FUNCTION_BLOCK "CompValEqOr"   // FB55, LAD
TITLE = COMP_VAL_==_OR_FB / COMP_VAL_==_OR
AUTHOR : SICAR
FAMILY : Miscellaneous
VERSION : 1.0
// Der Baustein vergleicht die Werte der Eingänge in1...in8 mit dem Wert des Eingangs „compareValue“ und verodert diese Vergleiche. Ist mindestens einer der Werte von in1...in8 gleich mit „compareValue“, so wird der Wert von „compareValue“ in den Output „value“ geschrieben. Andernfalls wird er mit dem Wert 0 beschrieben.  
// Anwendungsfall Beispiel: Damit kann ein "Summensignal" gebildet werden, z.B. für Produktionsdaten "Grenzwerte", womit ein Button animiert werden kann (Button "ProdData", "Grenzwerte").  
// 
// **Beispielaufruf**  
// Abbildung in Kontaktplan (KOP), ohne Parameterbeschaltung.  
// 
// **Aufrufschnittstelle**  
// Der Baustein wird im zyklischen Programm aufgerufen. In den Startup-Projekten ist der Baustein aufgerufen, für die Bildung eines Sammelsignals für die Grenzwerte der Produktionsdaten. Damit werden die Buttons  [ProdData]
// Compare the values of the inputs with the value of th input _compareValue_ generating a collective OR signal from these comparisons.
// stored: IsIECCheckEnabled true, MemoryReserve 100, SetENOAutomatically true
   VAR_INPUT
      compareValue { ExternalAccessible := 'False'; ExternalVisible := 'False'; ExternalWritable := 'False'} : UInt;   // Vergleichs Wert / Compare value
      val1 { ExternalAccessible := 'False'; ExternalVisible := 'False'; ExternalWritable := 'False'} : UInt;   // Wert 1 / value 1
      val2 { ExternalAccessible := 'False'; ExternalVisible := 'False'; ExternalWritable := 'False'} : UInt;   // Wert 2 / value 2
      val3 { ExternalAccessible := 'False'; ExternalVisible := 'False'; ExternalWritable := 'False'} : UInt;   // Wert 3 / value 3
      val4 { ExternalAccessible := 'False'; ExternalVisible := 'False'; ExternalWritable := 'False'} : UInt;   // Wert 4 / value 4
      val5 { ExternalAccessible := 'False'; ExternalVisible := 'False'; ExternalWritable := 'False'} : UInt;   // Wert 5 / value 5
      val6 { ExternalAccessible := 'False'; ExternalVisible := 'False'; ExternalWritable := 'False'} : UInt;   // Wert 6 / value 6
      val7 { ExternalAccessible := 'False'; ExternalVisible := 'False'; ExternalWritable := 'False'} : UInt;   // Wert 7 / value 7
      val8 { ExternalAccessible := 'False'; ExternalVisible := 'False'; ExternalWritable := 'False'} : UInt;   // Wert 8 / value 8
   END_VAR
   VAR_OUTPUT
      value { ExternalAccessible := 'False'; ExternalVisible := 'False'; ExternalWritable := 'False'} : UInt;   // Ergebnis Wert / Result value
   END_VAR
   VAR_TEMP
      tempDummy : Bool;   // Dummy
   END_VAR
BEGIN

REGION Network 1: Aufruf: Initialisierung SPS / ChangeLog
   // SIEMENS AG / (c)Copyright 2023
   // ------------------------------------------------------------------------------
   // Title:            CompValEqOr (FB55)
   // Comment/Function: Compare the values of the inputs with the value of th input compareValue generating a collective OR signal from these comparisons.
   // Library/Family:   Automation Framework
   // Author:           Siemens Digital Industry
   // Tested with:      ---
   // Engineering:      TIA Portal V19
   // Restrictions:     -
   // Requirements:     ---
   // ------------------------------------------------------------------------------
   // Change log table:
   // Version  | Date       | Expert in charge       | Changes applied
   // ---------|------------|------------------------|------------------------------
   // 01.00.00 | 11.12.2023 | Siemens Industry Online Support
   //                         First released version
END_REGION

REGION Network 2: Beschreibung / Description
   // The block compares the values of the inputs _in1 ... in8_ with the value of the input _compareValue_ and generates a collective OR signal from these comparisons. If at least one of the values of in1 ... in8 is equal with _compareValue_, the value of _compareValue_ is written to output “value”.  
   // Otherwise, “value” is written with the value 0.  
   // Use Case example: With this, a "summary signal" can be formed, e.g. for production data "Limit Values", with which a button can be animated (Button "ProdData", "LimitValues"). 
   // 
   // **Block call example**  
   // 
   // The call is shown as “Ladder Diagram” (LAD), without parameters.  
   // 
   // **Calling interface**  
   // 
   // The block is called in the cyclic program. In the startup projects, the block is called to generate a collective signal for the limit values of the production data. The buttons [ProdData] and [LimitValues] are animated in color, depending on the value range of the limit values.
   // 
   // **Operation mode Automatic / Manual**  
   // 
   // The block is independent of operation modes. Therefor it is not assigned to any operation mode area.
END_REGION

REGION Network 3: VALUE = 0 schreiben / set VALUE = 0
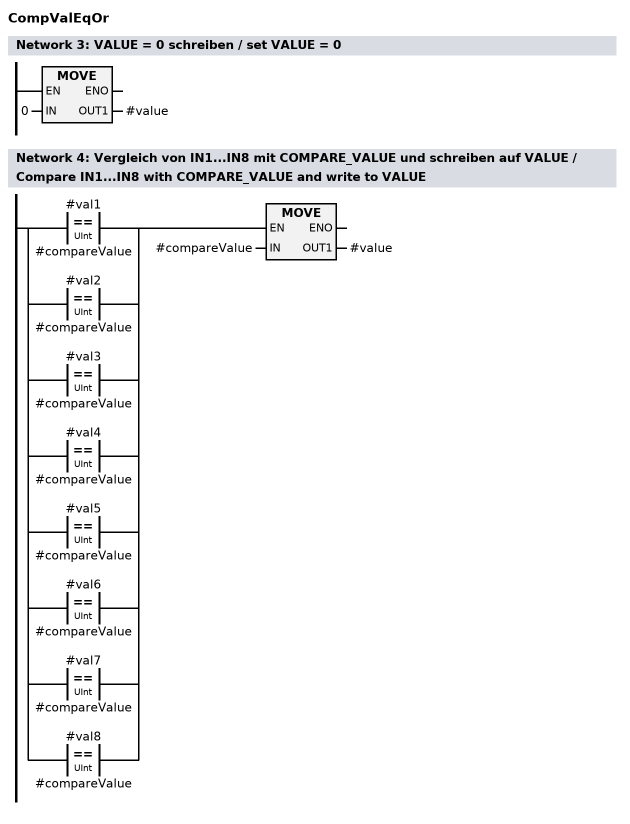
   RUNG wire#powerrail
      Move(in := 0, out1 => #value)
   END_RUNG
   // the same network as SCL:
   #value := 0;
END_REGION

REGION Network 4: Vergleich von IN1...IN8 mit COMPARE_VALUE und schreiben auf VALUE / Compare IN1...IN8 with COMPARE_VALUE and write to VALUE
   RUNG wire#powerrail
      { S7_Templates := "SrcType := UInt" } EQ_Contact(in1 := #val1, in2 := #compareValue)
      wire#w1
      Move(in := #compareValue, out1 => #value)
   END_RUNG
   RUNG wire#powerrail
      { S7_Templates := "SrcType := UInt" } EQ_Contact(in1 := #val2, in2 := #compareValue)
   END_RUNG wire#w1
   RUNG wire#powerrail
      { S7_Templates := "SrcType := UInt" } EQ_Contact(in1 := #val3, in2 := #compareValue)
   END_RUNG wire#w1
   RUNG wire#powerrail
      { S7_Templates := "SrcType := UInt" } EQ_Contact(in1 := #val4, in2 := #compareValue)
   END_RUNG wire#w1
   RUNG wire#powerrail
      { S7_Templates := "SrcType := UInt" } EQ_Contact(in1 := #val5, in2 := #compareValue)
   END_RUNG wire#w1
   RUNG wire#powerrail
      { S7_Templates := "SrcType := UInt" } EQ_Contact(in1 := #val6, in2 := #compareValue)
   END_RUNG wire#w1
   RUNG wire#powerrail
      { S7_Templates := "SrcType := UInt" } EQ_Contact(in1 := #val7, in2 := #compareValue)
   END_RUNG wire#w1
   RUNG wire#powerrail
      { S7_Templates := "SrcType := UInt" } EQ_Contact(in1 := #val8, in2 := #compareValue)
   END_RUNG wire#w1
   // the same network as SCL:
   IF (#val1 = #compareValue) OR (#val2 = #compareValue) OR (#val3 = #compareValue) OR (#val4 = #compareValue) OR (#val5 = #compareValue) OR (#val6 = #compareValue) OR (#val7 = #compareValue) OR (#val8 = #compareValue) THEN
       #value := #compareValue;
   END_IF;
END_REGION
END_FUNCTION_BLOCK

FUNCTION_BLOCK "CallAlarmCounter"   // FB5, LAD
// stored: MemoryReserve 100, SetENOAutomatically false
   VAR
      statPulse { ExternalAccessible := 'False'; ExternalVisible := 'False'; ExternalWritable := 'False'} : Array[0..99] of Bool;
   END_VAR
   VAR_TEMP
      tempEnter : Bool;   // Enter the conditions for the count to increase.
   END_VAR
   VAR_TEMP   // added for the SCL form of the ladder/FBD networks
      _w1 : Bool;
   END_VAR
BEGIN

REGION Network 1: Counter Setting Save
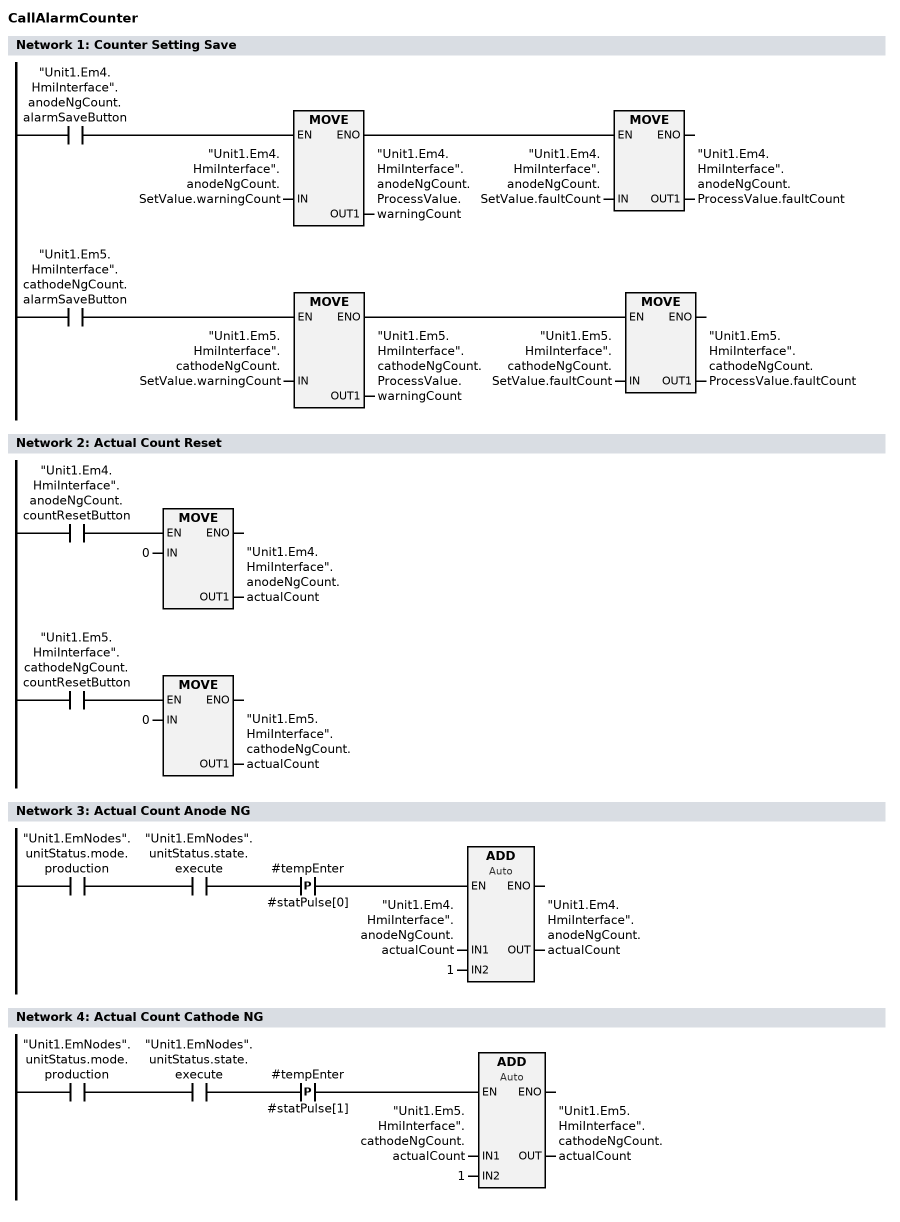
   RUNG wire#powerrail
      Contact( "Unit1.Em4.HmiInterface".anodeNgCount.alarmSaveButton )
      Move(in := "Unit1.Em4.HmiInterface".anodeNgCount.SetValue.warningCount, out1 => "Unit1.Em4.HmiInterface".anodeNgCount.ProcessValue.warningCount)
      Move(in := "Unit1.Em4.HmiInterface".anodeNgCount.SetValue.faultCount, out1 => "Unit1.Em4.HmiInterface".anodeNgCount.ProcessValue.faultCount)
   END_RUNG
   RUNG wire#powerrail
      Contact( "Unit1.Em5.HmiInterface".cathodeNgCount.alarmSaveButton )
      Move(in := "Unit1.Em5.HmiInterface".cathodeNgCount.SetValue.warningCount, out1 => "Unit1.Em5.HmiInterface".cathodeNgCount.ProcessValue.warningCount)
      Move(in := "Unit1.Em5.HmiInterface".cathodeNgCount.SetValue.faultCount, out1 => "Unit1.Em5.HmiInterface".cathodeNgCount.ProcessValue.faultCount)
   END_RUNG
   // the same network as SCL:
   IF "Unit1.Em4.HmiInterface".anodeNgCount.alarmSaveButton THEN
       "Unit1.Em4.HmiInterface".anodeNgCount.ProcessValue.warningCount := "Unit1.Em4.HmiInterface".anodeNgCount.SetValue.warningCount;
       "Unit1.Em4.HmiInterface".anodeNgCount.ProcessValue.faultCount := "Unit1.Em4.HmiInterface".anodeNgCount.SetValue.faultCount;
   END_IF;
   IF "Unit1.Em5.HmiInterface".cathodeNgCount.alarmSaveButton THEN
       "Unit1.Em5.HmiInterface".cathodeNgCount.ProcessValue.warningCount := "Unit1.Em5.HmiInterface".cathodeNgCount.SetValue.warningCount;
       "Unit1.Em5.HmiInterface".cathodeNgCount.ProcessValue.faultCount := "Unit1.Em5.HmiInterface".cathodeNgCount.SetValue.faultCount;
   END_IF;
END_REGION

REGION Network 2: Actual Count Reset
   RUNG wire#powerrail
      Contact( "Unit1.Em4.HmiInterface".anodeNgCount.countResetButton )
      Move(in := 0, out1 => "Unit1.Em4.HmiInterface".anodeNgCount.actualCount)
   END_RUNG
   RUNG wire#powerrail
      Contact( "Unit1.Em5.HmiInterface".cathodeNgCount.countResetButton )
      Move(in := 0, out1 => "Unit1.Em5.HmiInterface".cathodeNgCount.actualCount)
   END_RUNG
   // the same network as SCL:
   IF "Unit1.Em4.HmiInterface".anodeNgCount.countResetButton THEN
       "Unit1.Em4.HmiInterface".anodeNgCount.actualCount := 0;
   END_IF;
   IF "Unit1.Em5.HmiInterface".cathodeNgCount.countResetButton THEN
       "Unit1.Em5.HmiInterface".cathodeNgCount.actualCount := 0;
   END_IF;
END_REGION

REGION Network 3: Actual Count Anode NG
   RUNG wire#powerrail
      Contact( "Unit1.EmNodes".unitStatus.mode.production )
      Contact( "Unit1.EmNodes".unitStatus.state.execute )
      P_Contact(operand := #tempEnter, bit := #statPulse[0])
      Add(in1 := "Unit1.Em4.HmiInterface".anodeNgCount.actualCount, in2 := 1, out => "Unit1.Em4.HmiInterface".anodeNgCount.actualCount)
   END_RUNG
   // the same network as SCL:
   #_w1 := "Unit1.EmNodes".unitStatus.mode.production AND "Unit1.EmNodes".unitStatus.state.execute AND #tempEnter AND NOT #statPulse[0];   // rising edge of #tempEnter
   #statPulse[0] := #tempEnter;
   IF #_w1 THEN
       "Unit1.Em4.HmiInterface".anodeNgCount.actualCount := "Unit1.Em4.HmiInterface".anodeNgCount.actualCount + 1;
   END_IF;
END_REGION

REGION Network 4: Actual Count Cathode NG
   RUNG wire#powerrail
      Contact( "Unit1.EmNodes".unitStatus.mode.production )
      Contact( "Unit1.EmNodes".unitStatus.state.execute )
      P_Contact(operand := #tempEnter, bit := #statPulse[1])
      Add(in1 := "Unit1.Em5.HmiInterface".cathodeNgCount.actualCount, in2 := 1, out => "Unit1.Em5.HmiInterface".cathodeNgCount.actualCount)
   END_RUNG
   // the same network as SCL:
   #_w1 := "Unit1.EmNodes".unitStatus.mode.production AND "Unit1.EmNodes".unitStatus.state.execute AND #tempEnter AND NOT #statPulse[1];   // rising edge of #tempEnter
   #statPulse[1] := #tempEnter;
   IF #_w1 THEN
       "Unit1.Em5.HmiInterface".cathodeNgCount.actualCount := "Unit1.Em5.HmiInterface".cathodeNgCount.actualCount + 1;
   END_IF;
END_REGION
END_FUNCTION_BLOCK

FUNCTION "CallSettings" : Void   // FC8, LAD
// Call of settings blocks
// stored: IsIECCheckEnabled true, SetENOAutomatically false
BEGIN

REGION Network 1: Beschreibung / BLOCK INFO HEADER
   // **Betriebsart Automatik / Hand**  
   // Der Baustein ist keiner Betriebsart / Betriebsartenbereich zugeordnet.  
   // 
   // **Alarme**  
   // Der Baustein generiert keine Alarme.  
   // 
   // #### PLC-Datentypen  
   // Verwendete PLC-Datentypen für den SPS-Programmbaustein und das zugehörige WinCC-Bild.  
   // 
   // {.pageWidth}
   // ![Image](CallInterfaceSignals/de/image1.PNG)
   //  
   //  
   // #### Bausteinaufrufe 
   // Der Baustein “LSicar_InterfaceSignalsBool“ wird in diesem FB als Multi-Instanz aufgerufen, entspr. nebenstehender beispielhafter Darstellung.  
   // 
   // {.pageWidth}
   // ![Image](CallInterfaceSignals/de/image2.PNG)
   //  
   // Um einen neuen FB aufzurufen, ziehen Sie den FB in ein neues Netzwerk, wählen Sie „Multiinstanz“ aus, vergeben Sie einen Namen und parametrieren Sie den FB-Aufruf.  
   // 
   // {.pageWidth}
   // ![Image](CallInterfaceSignals/de/image3.PNG)
   //  
   //  
   // #### Weitere Hinweise 
   // 
   // #### Updateinfo 
   // 
   // #### Weitere Dokumente 
   // 
   // ![Icon](_Icon/reference.PNG)
   // 
   // ..\Library Types\LSicar_InterfaceSignalsBool.pdf
   // SIEMENS AG / (c)Copyright 2023
   // ------------------------------------------------------------------------------
   // Title:            CallSettings
   // Comment/Function: Call of SICAR Settings blocks
   // Library/Family:   -
   // Author:           -
   // Tested with:      ---
   // Engineering:      TIA Portal V19
   // Restrictions:     -
   // Requirements:     ---
   // ------------------------------------------------------------------------------
   // Change log table:
   // Version | Date | Expert in charge | Changes applied
   // -------|---------|-------------|--------------------------------------------
   // 01.00.00 | 01.01.1999 | Person x | First released version
   // 01.00.01 | 02.01.1999 | Person y | Block was Updated
END_REGION

REGION Network 2: Set set PLC date and time
   // Change local date and time of the PLC
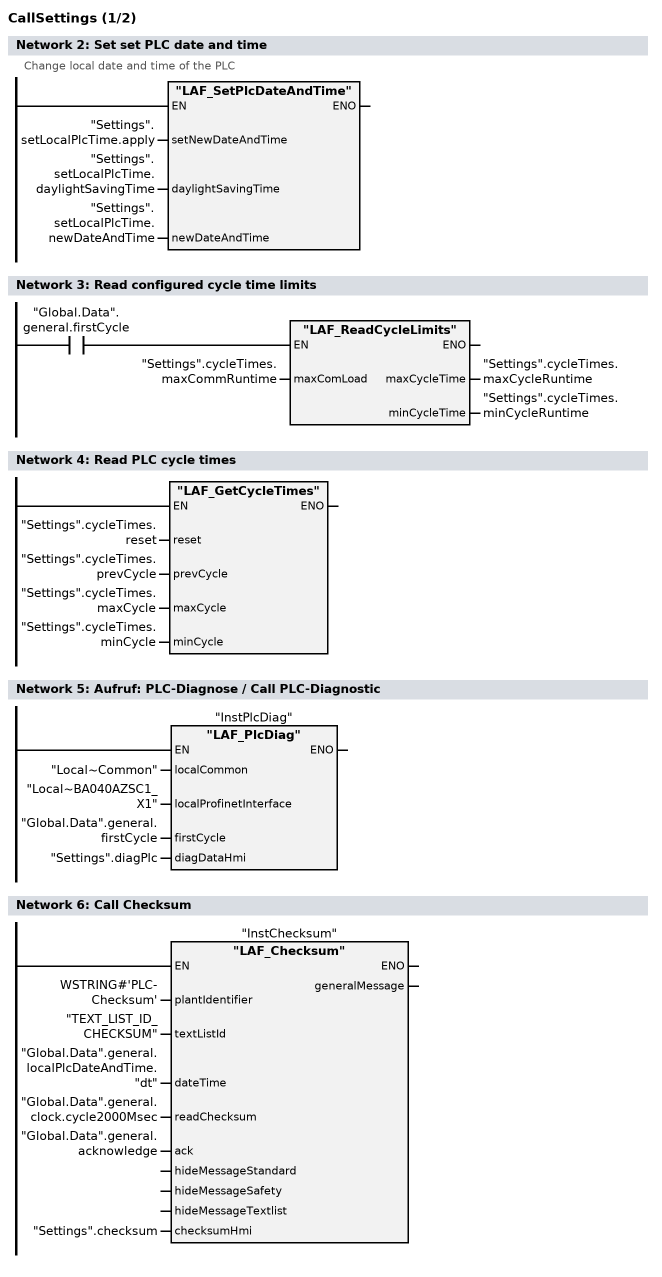
   RUNG wire#powerrail
      "LAF_SetPlcDateAndTime"(setNewDateAndTime := "Settings".setLocalPlcTime.apply, daylightSavingTime := "Settings".setLocalPlcTime.daylightSavingTime, newDateAndTime := "Settings".setLocalPlcTime.newDateAndTime)
   END_RUNG
   // the same network as SCL:
   "LAF_SetPlcDateAndTime"(setNewDateAndTime := "Settings".setLocalPlcTime.apply,
                           daylightSavingTime := "Settings".setLocalPlcTime.daylightSavingTime,
                           newDateAndTime := "Settings".setLocalPlcTime.newDateAndTime);
END_REGION

REGION Network 3: Read configured cycle time limits
   RUNG wire#powerrail
      Contact( "Global.Data".general.firstCycle )
      "LAF_ReadCycleLimits"(maxComLoad := "Settings".cycleTimes.maxCommRuntime, maxCycleTime => "Settings".cycleTimes.maxCycleRuntime, minCycleTime => "Settings".cycleTimes.minCycleRuntime)
   END_RUNG
   // the same network as SCL:
   IF "Global.Data".general.firstCycle THEN
       "LAF_ReadCycleLimits"(maxComLoad := "Settings".cycleTimes.maxCommRuntime,
                             maxCycleTime => "Settings".cycleTimes.maxCycleRuntime,
                             minCycleTime => "Settings".cycleTimes.minCycleRuntime);
   END_IF;
END_REGION

REGION Network 4: Read PLC cycle times
   RUNG wire#powerrail
      "LAF_GetCycleTimes"(reset := "Settings".cycleTimes.reset, prevCycle := "Settings".cycleTimes.prevCycle, maxCycle := "Settings".cycleTimes.maxCycle, minCycle := "Settings".cycleTimes.minCycle)
   END_RUNG
   // the same network as SCL:
   "LAF_GetCycleTimes"(reset := "Settings".cycleTimes.reset,
                       prevCycle := "Settings".cycleTimes.prevCycle,
                       maxCycle := "Settings".cycleTimes.maxCycle,
                       minCycle := "Settings".cycleTimes.minCycle);
END_REGION

REGION Network 5: Aufruf: PLC-Diagnose / Call PLC-Diagnostic
   RUNG wire#powerrail
      "InstPlcDiag"(localCommon := "Local~Common", localProfinetInterface := "Local~BA040AZSC1_X1", firstCycle := "Global.Data".general.firstCycle, diagDataHmi := "Settings".diagPlc)
   END_RUNG
   // the same network as SCL:
   "InstPlcDiag"(localCommon := "Local~Common",   // "LAF_PlcDiag"
                 localProfinetInterface := "Local~BA040AZSC1_X1",
                 firstCycle := "Global.Data".general.firstCycle,
                 diagDataHmi := "Settings".diagPlc);
END_REGION

REGION Network 6: Call Checksum
   RUNG wire#powerrail
      "InstChecksum"(plantIdentifier := WSTRING#'PLC-Checksum', textListId := "TEXT_LIST_ID_CHECKSUM", dateTime := "Global.Data".general.localPlcDateAndTime."dt", readChecksum := "Global.Data".general.clock.cycle2000Msec, ack := "Global.Data".general.acknowledge, hideMessageStandard :=, hideMessageSafety :=, hideMessageTextlist :=, checksumHmi := "Settings".checksum, generalMessage =>)
   END_RUNG
   // the same network as SCL:
   "InstChecksum"(plantIdentifier := WSTRING#'PLC-Checksum',   // "LAF_Checksum"
                  textListId := "TEXT_LIST_ID_CHECKSUM",
                  dateTime := "Global.Data".general.localPlcDateAndTime."dt",
                  readChecksum := "Global.Data".general.clock.cycle2000Msec,
                  ack := "Global.Data".general.acknowledge,
                  checksumHmi := "Settings".checksum);
END_REGION

REGION Network 7: Aufruf: SMC-Diagnose (SIMATIC Memory Card - Diagnose) / Call SMC-Diagnostic (SIMATIC Memory Card - Diagnostic)
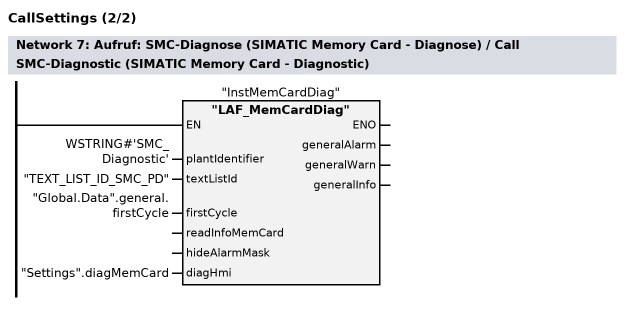
   RUNG wire#powerrail
      "InstMemCardDiag"(plantIdentifier := WSTRING#'SMC_Diagnostic', textListId := "TEXT_LIST_ID_SMC_PD", firstCycle := "Global.Data".general.firstCycle, readInfoMemCard :=, hideAlarmMask :=, diagHmi := "Settings".diagMemCard, generalAlarm =>, generalWarn =>, generalInfo =>)
   END_RUNG
   // the same network as SCL:
   "InstMemCardDiag"(plantIdentifier := WSTRING#'SMC_Diagnostic',   // "LAF_MemCardDiag"
                     textListId := "TEXT_LIST_ID_SMC_PD",
                     firstCycle := "Global.Data".general.firstCycle,
                     diagHmi := "Settings".diagMemCard);
END_REGION
END_FUNCTION

FUNCTION "CallEnergy" : Void   // FC5, LAD
TITLE = CallEnergy
// Call of Demo EnergyMeter and Energy Efficient M for EEMM demonstration
// stored: IsIECCheckEnabled true, SetENOAutomatically true
BEGIN

REGION Network 1: BLOCK INFO HEADER
   // SIEMENS AG / (c)Copyright 2023
   // ------------------------------------------------------------------------------
   // Title:            CallEnergy (FC5)
   // Comment/Function: Call of Demo EnergyMeter and Energy Efficient M for EEMM demonstration
   // Library/Family:   Energy
   // Author:           SICAR
   // Tested with:      ---
   // Engineering:      TIA Portal V19
   // Restrictions:     -
   // Requirements:     ---
   // ------------------------------------------------------------------------------
   // Change log table:
   // Version  | Date       | Expert in charge       | Changes applied
   // ---------|------------|------------------------|------------------------------
   // 01.00.00 | 11.12.2023 | SICAR
   //                         First released version
END_REGION

REGION Network 2: Call: Demo EnergyMeter, Energy Efficient M
   // Call for EEM demonstration
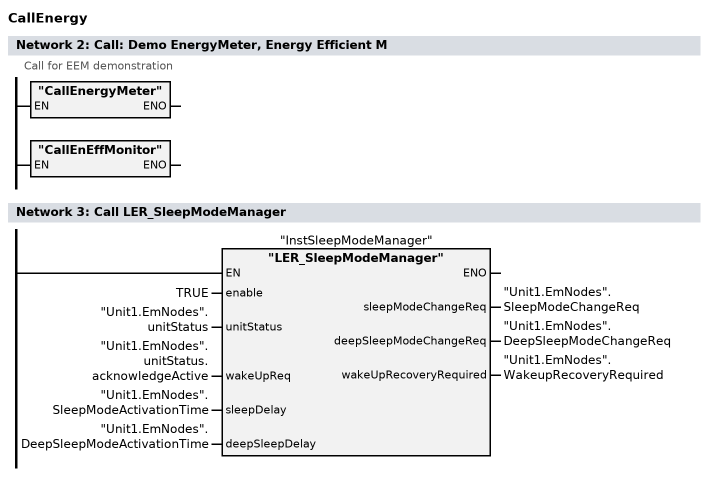
   RUNG wire#powerrail
      "CallEnergyMeter"()
   END_RUNG
   RUNG wire#powerrail
      "CallEnEffMonitor"()
   END_RUNG
   // the same network as SCL:
   "CallEnergyMeter"();
   "CallEnEffMonitor"();
END_REGION

REGION Network 3: Call LER_SleepModeManager
   RUNG wire#powerrail
      "InstSleepModeManager"(enable := TRUE, unitStatus := "Unit1.EmNodes".unitStatus, wakeUpReq := "Unit1.EmNodes".unitStatus.acknowledgeActive, sleepDelay := "Unit1.EmNodes".SleepModeActivationTime, deepSleepDelay := "Unit1.EmNodes".DeepSleepModeActivationTime, sleepModeChangeReq => "Unit1.EmNodes".SleepModeChangeReq, deepSleepModeChangeReq => "Unit1.EmNodes".DeepSleepModeChangeReq, wakeUpRecoveryRequired => "Unit1.EmNodes".WakeupRecoveryRequired)
   END_RUNG
   // the same network as SCL:
   "InstSleepModeManager"(enable := TRUE,   // "LER_SleepModeManager"
                          unitStatus := "Unit1.EmNodes".unitStatus,
                          wakeUpReq := "Unit1.EmNodes".unitStatus.acknowledgeActive,
                          sleepDelay := "Unit1.EmNodes".SleepModeActivationTime,
                          deepSleepDelay := "Unit1.EmNodes".DeepSleepModeActivationTime,
                          sleepModeChangeReq => "Unit1.EmNodes".SleepModeChangeReq,
                          deepSleepModeChangeReq => "Unit1.EmNodes".DeepSleepModeChangeReq,
                          wakeUpRecoveryRequired => "Unit1.EmNodes".WakeupRecoveryRequired);
END_REGION
END_FUNCTION

FUNCTION "CallEnergyMeter" : Void   // FC9, LAD
TITLE = CALL_AIEnergyMeter_FC
AUTHOR : SICAR
FAMILY : Energy
VERSION : 1.0
// FUNKTIONSBESCHREIBUNG: 
// Der Baustein dient als Aufrufschnittstelle für die bausteine des AI-Energy-Managements.
// Weitere Hinweise: siehe SICAR anwenderdefinierte Dokumentation / SICAR Online-Hilfe.
// This block calls the blocks for the AI-Energy-management.
// For more informations see SICAR userdefined documentation / SICAR online-help.
// stored: IsIECCheckEnabled true, SetENOAutomatically true
   VAR_TEMP
      tempCommResourceCounter : Int;   // für FB-Aufruf: E2M_1500_AIEnergyMeter_DRV
      tempBitsHmi : "typeEnMeterBits";   // für FB-Aufruf: E2M_1500_AIEnergyMeter_DRV
   END_VAR
   // Ret_Val : Ret_Val
BEGIN

REGION Network 1: Änderungshistorie / ChangeLog
   // Die Änderungshistorie wird nur in englischer Editiersprache geführt.
   // SIEMENS AG / (c)Copyright 2023
   // ------------------------------------------------------------------------------
   // Title:            CallEnergyMeter (FC9)
   // Comment/Function: This block calls the blocks for the AI-Energy-management.
   // Library/Family:   Automation Framework
   // Author:           Siemens Digital Industry
   // Tested with:      ---
   // Engineering:      TIA Portal V19
   // Restrictions:     -
   // Requirements:     ---
   // ------------------------------------------------------------------------------
   // Change log table:
   // Version  | Date       | Expert in charge       | Changes applied
   // ---------|------------|------------------------|------------------------------
   // 05.00.00 | 01.09.2023 | SICAR
   //                         First released version
END_REGION

REGION Network 2: AI_EnergyMeter 1
   // Aufruf von E2MenergyMeterDrv FB / Call of E2MenergyMeterDrv FB
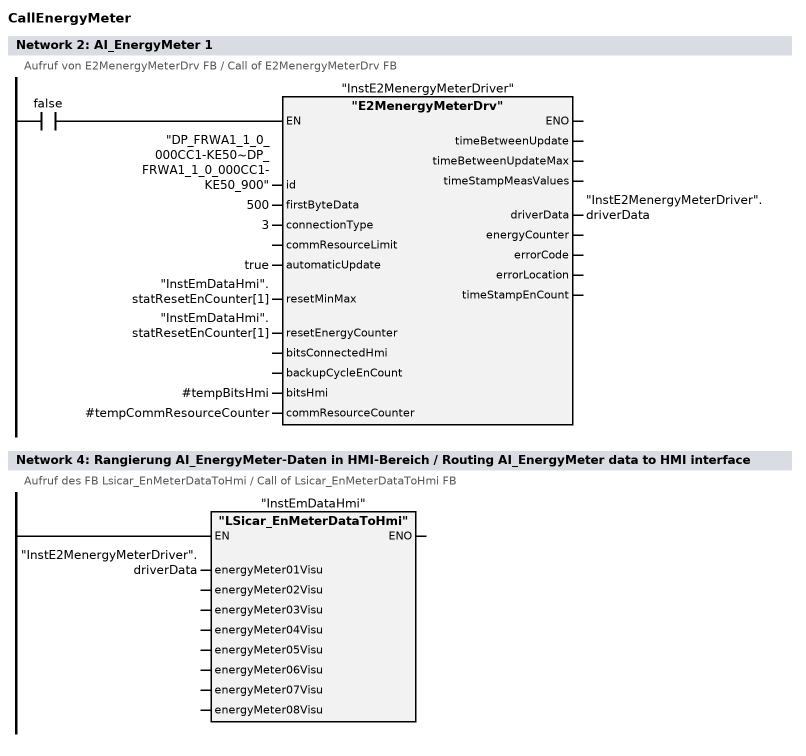
   RUNG wire#powerrail
      Contact( false )
      "InstE2MenergyMeterDriver"(id := "DP_FRWA1_1_0_000CC1-KE50~DP_FRWA1_1_0_000CC1-KE50_900", firstByteData := 500, connectionType := 3, commResourceLimit :=, automaticUpdate := true, resetMinMax := "InstEmDataHmi".statResetEnCounter[1], resetEnergyCounter := "InstEmDataHmi".statResetEnCounter[1], bitsConnectedHmi :=, backupCycleEnCount :=, bitsHmi := #tempBitsHmi, commResourceCounter := #tempCommResourceCounter, timeBetweenUpdate =>, timeBetweenUpdateMax =>, timeStampMeasValues =>, driverData => "InstE2MenergyMeterDriver".driverData, energyCounter =>, errorCode =>, errorLocation =>, timeStampEnCount =>)
   END_RUNG
   // the same network as SCL:
   IF false THEN
       "InstE2MenergyMeterDriver"(id := "DP_FRWA1_1_0_000CC1-KE50~DP_FRWA1_1_0_000CC1-KE50_900",   // "E2MenergyMeterDrv"
                               firstByteData := 500,
                               connectionType := 3,
                               automaticUpdate := true,
                               resetMinMax := "InstEmDataHmi".statResetEnCounter[1],
                               resetEnergyCounter := "InstEmDataHmi".statResetEnCounter[1],
                               bitsHmi := #tempBitsHmi,
                               commResourceCounter := #tempCommResourceCounter,
                               driverData => "InstE2MenergyMeterDriver".driverData);
   END_IF;
END_REGION

REGION Network 3 (SCL): Power meter

   // Voltage L-N
   "InstE2MenergyMeterDriver".driverData.uL1 := "PAC3220InPut"."Voltage_L1-N";
   "InstE2MenergyMeterDriver".driverData.uL2 := "PAC3220InPut"."Voltage_L2-N";
   "InstE2MenergyMeterDriver".driverData.uL3 := "PAC3220InPut"."Voltage_L3-N";
   "InstE2MenergyMeterDriver".driverData.uPhNaverage :=
   ("InstE2MenergyMeterDriver".driverData.uL1 + "InstE2MenergyMeterDriver".driverData.uL2 + "InstE2MenergyMeterDriver".driverData.uL3) / 3.0;

   IF "InstE2MenergyMeterDriver".driverData.uL1 < "InstE2MenergyMeterDriver".driverData.uL1Min OR "InstE2MenergyMeterDriver".driverData.uL1Min = 0.0 THEN
       "InstE2MenergyMeterDriver".driverData.uL1Min := "InstE2MenergyMeterDriver".driverData.uL1;
   END_IF;
   IF "InstE2MenergyMeterDriver".driverData.uL1 > "InstE2MenergyMeterDriver".driverData.uL1Max OR "InstE2MenergyMeterDriver".driverData.uL1Max = 0.0 THEN
       "InstE2MenergyMeterDriver".driverData.uL1Max := "InstE2MenergyMeterDriver".driverData.uL1;
   END_IF;

   IF "InstE2MenergyMeterDriver".driverData.uL2 < "InstE2MenergyMeterDriver".driverData.uL2Min OR "InstE2MenergyMeterDriver".driverData.uL2Min = 0.0 THEN
       "InstE2MenergyMeterDriver".driverData.uL2Min := "InstE2MenergyMeterDriver".driverData.uL2;
   END_IF;
   IF "InstE2MenergyMeterDriver".driverData.uL2 > "InstE2MenergyMeterDriver".driverData.uL2Max OR "InstE2MenergyMeterDriver".driverData.uL2Max = 0.0 THEN
       "InstE2MenergyMeterDriver".driverData.uL2Max := "InstE2MenergyMeterDriver".driverData.uL2;
   END_IF;

   IF "InstE2MenergyMeterDriver".driverData.uL3 < "InstE2MenergyMeterDriver".driverData.uL3Min OR "InstE2MenergyMeterDriver".driverData.uL3Min = 0.0 THEN
       "InstE2MenergyMeterDriver".driverData.uL3Min := "InstE2MenergyMeterDriver".driverData.uL3;
   END_IF;
   IF "InstE2MenergyMeterDriver".driverData.uL3 > "InstE2MenergyMeterDriver".driverData.uL3Max OR "InstE2MenergyMeterDriver".driverData.uL3Max = 0.0 THEN
       "InstE2MenergyMeterDriver".driverData.uL3Max := "InstE2MenergyMeterDriver".driverData.uL3;
   END_IF;

   IF "InstE2MenergyMeterDriver".driverData.uPhNaverage < "InstE2MenergyMeterDriver".driverData.uPhNaverageMin OR "InstE2MenergyMeterDriver".driverData.uPhNaverageMin = 0.0 THEN
       "InstE2MenergyMeterDriver".driverData.uPhNaverageMin := "InstE2MenergyMeterDriver".driverData.uPhNaverage;
   END_IF;
   IF "InstE2MenergyMeterDriver".driverData.uPhNaverage > "InstE2MenergyMeterDriver".driverData.uPhNaverageMax OR "InstE2MenergyMeterDriver".driverData.uPhNaverageMax = 0.0 THEN
       "InstE2MenergyMeterDriver".driverData.uPhNaverageMax := "InstE2MenergyMeterDriver".driverData.uPhNaverage;
   END_IF;

   // Voltage L-L
   "InstE2MenergyMeterDriver".driverData.uL1L2 := "PAC3220InPut"."Voltage_L1-L2";
   "InstE2MenergyMeterDriver".driverData.uL2L3 := "PAC3220InPut"."Voltage_L2-L3";
   "InstE2MenergyMeterDriver".driverData.uL3L1 := "PAC3220InPut"."Voltage_L3-L1";
   "InstE2MenergyMeterDriver".driverData.uPhPhAverage :=
   ("InstE2MenergyMeterDriver".driverData.uL1L2 + "InstE2MenergyMeterDriver".driverData.uL2L3 + "InstE2MenergyMeterDriver".driverData.uL3L1) / 3.0;

   IF "InstE2MenergyMeterDriver".driverData.uL1L2 < "InstE2MenergyMeterDriver".driverData.uL1L2Min OR "InstE2MenergyMeterDriver".driverData.uL1L2Min = 0.0 THEN
       "InstE2MenergyMeterDriver".driverData.uL1L2Min := "InstE2MenergyMeterDriver".driverData.uL1L2;
   END_IF;
   IF "InstE2MenergyMeterDriver".driverData.uL1L2 > "InstE2MenergyMeterDriver".driverData.uL1L2Max OR "InstE2MenergyMeterDriver".driverData.uL1L2Max = 0.0 THEN
       "InstE2MenergyMeterDriver".driverData.uL1L2Max := "InstE2MenergyMeterDriver".driverData.uL1L2;
   END_IF;

   IF "InstE2MenergyMeterDriver".driverData.uL2L3 < "InstE2MenergyMeterDriver".driverData.uL2L3Min OR "InstE2MenergyMeterDriver".driverData.uL2L3Min = 0.0 THEN
       "InstE2MenergyMeterDriver".driverData.uL2L3Min := "InstE2MenergyMeterDriver".driverData.uL2L3;
   END_IF;
   IF "InstE2MenergyMeterDriver".driverData.uL2L3 > "InstE2MenergyMeterDriver".driverData.uL2L3Max OR "InstE2MenergyMeterDriver".driverData.uL2L3Max = 0.0 THEN
       "InstE2MenergyMeterDriver".driverData.uL2L3Max := "InstE2MenergyMeterDriver".driverData.uL2L3;
   END_IF;

   IF "InstE2MenergyMeterDriver".driverData.uL3L1 < "InstE2MenergyMeterDriver".driverData.uL3L1Min OR "InstE2MenergyMeterDriver".driverData.uL3L1Min = 0.0 THEN
       "InstE2MenergyMeterDriver".driverData.uL3L1Min := "InstE2MenergyMeterDriver".driverData.uL3L1;
   END_IF;
   IF "InstE2MenergyMeterDriver".driverData.uL3L1 > "InstE2MenergyMeterDriver".driverData.uL3L1Max OR "InstE2MenergyMeterDriver".driverData.uL3L1Max = 0.0 THEN
       "InstE2MenergyMeterDriver".driverData.uL3L1Max := "InstE2MenergyMeterDriver".driverData.uL3L1;
   END_IF;

   IF "InstE2MenergyMeterDriver".driverData.uPhPhAverage < "InstE2MenergyMeterDriver".driverData.uPhPhAverageMin OR "InstE2MenergyMeterDriver".driverData.uPhPhAverageMin = 0.0 THEN
       "InstE2MenergyMeterDriver".driverData.uPhPhAverageMin := "InstE2MenergyMeterDriver".driverData.uPhPhAverage;
   END_IF;
   IF "InstE2MenergyMeterDriver".driverData.uPhPhAverage > "InstE2MenergyMeterDriver".driverData.uPhPhAverageMax OR "InstE2MenergyMeterDriver".driverData.uPhPhAverageMax = 0.0THEN
       "InstE2MenergyMeterDriver".driverData.uPhPhAverageMax := "InstE2MenergyMeterDriver".driverData.uPhPhAverage;
   END_IF;

   // Current
   "InstE2MenergyMeterDriver".driverData.iL1 := "PAC3220InPut".Current_L1;
   "InstE2MenergyMeterDriver".driverData.iL2 := "PAC3220InPut".Current_L2;
   "InstE2MenergyMeterDriver".driverData.iL3 := "PAC3220InPut".Current_L3;
   "InstE2MenergyMeterDriver".driverData.iAverage := "PAC3220InPut"."3-phase_average_current";

   IF "InstE2MenergyMeterDriver".driverData.iL1 < "InstE2MenergyMeterDriver".driverData.iL1Min OR "InstE2MenergyMeterDriver".driverData.iL1Min = 0.0 THEN
       "InstE2MenergyMeterDriver".driverData.iL1Min := "InstE2MenergyMeterDriver".driverData.iL1;
   END_IF;
   IF "InstE2MenergyMeterDriver".driverData.iL1 > "InstE2MenergyMeterDriver".driverData.iL1Max OR "InstE2MenergyMeterDriver".driverData.iL1Max = 0.0 THEN
       "InstE2MenergyMeterDriver".driverData.iL1Max := "InstE2MenergyMeterDriver".driverData.iL1;
   END_IF;

   IF "InstE2MenergyMeterDriver".driverData.iL2 < "InstE2MenergyMeterDriver".driverData.iL2Min OR "InstE2MenergyMeterDriver".driverData.iL2Min = 0.0 THEN
       "InstE2MenergyMeterDriver".driverData.iL2Min := "InstE2MenergyMeterDriver".driverData.iL2;
   END_IF;
   IF "InstE2MenergyMeterDriver".driverData.iL2 > "InstE2MenergyMeterDriver".driverData.iL2Max OR "InstE2MenergyMeterDriver".driverData.iL2Max = 0.0 THEN
       "InstE2MenergyMeterDriver".driverData.iL2Max := "InstE2MenergyMeterDriver".driverData.iL2;
   END_IF;

   IF "InstE2MenergyMeterDriver".driverData.iL3 < "InstE2MenergyMeterDriver".driverData.iL3Min OR "InstE2MenergyMeterDriver".driverData.iL3Min = 0.0 THEN
       "InstE2MenergyMeterDriver".driverData.iL3Min := "InstE2MenergyMeterDriver".driverData.iL3;
   END_IF;
   IF "InstE2MenergyMeterDriver".driverData.iL3 > "InstE2MenergyMeterDriver".driverData.iL3Max OR "InstE2MenergyMeterDriver".driverData.iL3Max = 0.0 THEN
       "InstE2MenergyMeterDriver".driverData.iL3Max := "InstE2MenergyMeterDriver".driverData.iL3;
   END_IF;

   IF "InstE2MenergyMeterDriver".driverData.iAverage < "InstE2MenergyMeterDriver".driverData.iAverageMin OR "InstE2MenergyMeterDriver".driverData.iAverageMin = 0.0 THEN
       "InstE2MenergyMeterDriver".driverData.iAverageMin := "InstE2MenergyMeterDriver".driverData.iAverage;
   END_IF;
   IF "InstE2MenergyMeterDriver".driverData.iAverage > "InstE2MenergyMeterDriver".driverData.iAverageMax OR "InstE2MenergyMeterDriver".driverData.iAverageMax = 0.0THEN
       "InstE2MenergyMeterDriver".driverData.iAverageMax := "InstE2MenergyMeterDriver".driverData.iAverage;
   END_IF;

   // Power factor
   "InstE2MenergyMeterDriver".driverData.cosL1 := "PAC3220InPut".Power_factor_L1;
   "InstE2MenergyMeterDriver".driverData.cosL2 := "PAC3220InPut".Power_factor_L2;
   "InstE2MenergyMeterDriver".driverData.cosL3 := "PAC3220InPut".Power_factor_L3;
   "InstE2MenergyMeterDriver".driverData.cosAverage := "PAC3220InPut".Total_power_factor;

   IF "InstE2MenergyMeterDriver".driverData.cosL1 < "InstE2MenergyMeterDriver".driverData.cosL1Min OR "InstE2MenergyMeterDriver".driverData.cosL1Min = 0.0 THEN
       "InstE2MenergyMeterDriver".driverData.cosL1Min := "InstE2MenergyMeterDriver".driverData.cosL1;
   END_IF;
   IF "InstE2MenergyMeterDriver".driverData.cosL1 > "InstE2MenergyMeterDriver".driverData.cosL1Max THEN
       "InstE2MenergyMeterDriver".driverData.cosL1Max := "InstE2MenergyMeterDriver".driverData.cosL1;
   END_IF;

   IF "InstE2MenergyMeterDriver".driverData.cosL2 < "InstE2MenergyMeterDriver".driverData.cosL2Min OR "InstE2MenergyMeterDriver".driverData.cosL2Min = 0.0 THEN
       "InstE2MenergyMeterDriver".driverData.cosL2Min := "InstE2MenergyMeterDriver".driverData.cosL2;
   END_IF;
   IF "InstE2MenergyMeterDriver".driverData.cosL2 > "InstE2MenergyMeterDriver".driverData.cosL2Max OR "InstE2MenergyMeterDriver".driverData.cosL2Max = 0.0 THEN
       "InstE2MenergyMeterDriver".driverData.cosL2Max := "InstE2MenergyMeterDriver".driverData.cosL2;
   END_IF;

   IF "InstE2MenergyMeterDriver".driverData.cosL3 < "InstE2MenergyMeterDriver".driverData.cosL3Min OR "InstE2MenergyMeterDriver".driverData.cosL3Min = 0.0 THEN
       "InstE2MenergyMeterDriver".driverData.cosL3Min := "InstE2MenergyMeterDriver".driverData.cosL3;
   END_IF;
   IF "InstE2MenergyMeterDriver".driverData.cosL3 > "InstE2MenergyMeterDriver".driverData.cosL3Max OR "InstE2MenergyMeterDriver".driverData.cosL3Max = 0.0THEN
       "InstE2MenergyMeterDriver".driverData.cosL3Max := "InstE2MenergyMeterDriver".driverData.cosL3;
   END_IF;

   IF "InstE2MenergyMeterDriver".driverData.cosAverage < "InstE2MenergyMeterDriver".driverData.cosAverageMin OR "InstE2MenergyMeterDriver".driverData.cosAverageMin = 0.0 THEN
       "InstE2MenergyMeterDriver".driverData.cosAverageMin := "InstE2MenergyMeterDriver".driverData.cosAverage;
   END_IF;
   IF "InstE2MenergyMeterDriver".driverData.cosAverage > "InstE2MenergyMeterDriver".driverData.cosAverageMax OR "InstE2MenergyMeterDriver".driverData.cosAverageMax = 0.0 THEN
       "InstE2MenergyMeterDriver".driverData.cosAverageMax := "InstE2MenergyMeterDriver".driverData.cosAverage;
   END_IF;

   // Frequency
   "InstE2MenergyMeterDriver".driverData.f := "PAC3220InPut".Line_frequency;

   IF "InstE2MenergyMeterDriver".driverData.f < "InstE2MenergyMeterDriver".driverData.fMin OR "InstE2MenergyMeterDriver".driverData.fMin = 0.0 THEN
       "InstE2MenergyMeterDriver".driverData.fMin := "InstE2MenergyMeterDriver".driverData.f;
   END_IF;
   IF "InstE2MenergyMeterDriver".driverData.f > "InstE2MenergyMeterDriver".driverData.fMax OR "InstE2MenergyMeterDriver".driverData.fMax = 0.0 THEN
       "InstE2MenergyMeterDriver".driverData.fMax := "InstE2MenergyMeterDriver".driverData.f;
   END_IF;


   // Apparent power
   "InstE2MenergyMeterDriver".driverData.sL1 := "Apparent power L1";
   "InstE2MenergyMeterDriver".driverData.sL2 := "Apparent power L2";
   "InstE2MenergyMeterDriver".driverData.sL3 := "Apparent power L3";
   "InstE2MenergyMeterDriver".driverData.sTotal := "PAC3220InPut".Total_apparent_power;

   IF "InstE2MenergyMeterDriver".driverData.sL1 < "InstE2MenergyMeterDriver".driverData.sL1Min OR "InstE2MenergyMeterDriver".driverData.sL1Min = 0.0 THEN
       "InstE2MenergyMeterDriver".driverData.sL1Min := "InstE2MenergyMeterDriver".driverData.sL1;
   END_IF;
   IF "InstE2MenergyMeterDriver".driverData.sL1 > "InstE2MenergyMeterDriver".driverData.sL1Max OR "InstE2MenergyMeterDriver".driverData.sL1Max = 0.0 THEN
       "InstE2MenergyMeterDriver".driverData.sL1Max := "InstE2MenergyMeterDriver".driverData.sL1;
   END_IF;

   IF "InstE2MenergyMeterDriver".driverData.sL2 < "InstE2MenergyMeterDriver".driverData.sL2Min OR "InstE2MenergyMeterDriver".driverData.sL2Min = 0.0 THEN
       "InstE2MenergyMeterDriver".driverData.sL2Min := "InstE2MenergyMeterDriver".driverData.sL2;
   END_IF;
   IF "InstE2MenergyMeterDriver".driverData.sL2 > "InstE2MenergyMeterDriver".driverData.sL2Max OR "InstE2MenergyMeterDriver".driverData.sL2Max = 0.0 THEN
       "InstE2MenergyMeterDriver".driverData.sL2Max := "InstE2MenergyMeterDriver".driverData.sL2;
   END_IF;

   IF "InstE2MenergyMeterDriver".driverData.sL3 < "InstE2MenergyMeterDriver".driverData.sL3Min OR "InstE2MenergyMeterDriver".driverData.sL3Min = 0.0 THEN
       "InstE2MenergyMeterDriver".driverData.sL3Min := "InstE2MenergyMeterDriver".driverData.sL3;
   END_IF;
   IF "InstE2MenergyMeterDriver".driverData.sL3 > "InstE2MenergyMeterDriver".driverData.sL3Max OR "InstE2MenergyMeterDriver".driverData.sL3Max = 0.0 THEN
       "InstE2MenergyMeterDriver".driverData.sL3Max := "InstE2MenergyMeterDriver".driverData.sL3;
   END_IF;

   IF "InstE2MenergyMeterDriver".driverData.sTotal < "InstE2MenergyMeterDriver".driverData.sTotalMin OR "InstE2MenergyMeterDriver".driverData.sTotalMin = 0.0 THEN
       "InstE2MenergyMeterDriver".driverData.sTotalMin := "InstE2MenergyMeterDriver".driverData.sTotal;
   END_IF;
   IF "InstE2MenergyMeterDriver".driverData.sTotal > "InstE2MenergyMeterDriver".driverData.sTotalMax OR "InstE2MenergyMeterDriver".driverData.sTotalMax = 0.0 THEN
       "InstE2MenergyMeterDriver".driverData.sTotalMax := "InstE2MenergyMeterDriver".driverData.sTotal;
   END_IF;

   // Active power
   "InstE2MenergyMeterDriver".driverData.pL1 := "Active power L1";
   "InstE2MenergyMeterDriver".driverData.pL2 := "Active power L2";
   "InstE2MenergyMeterDriver".driverData.pL3 := "Active power L3";
   "InstE2MenergyMeterDriver".driverData.pTotal := "PAC3220InPut".Total_active_power;

   IF "InstE2MenergyMeterDriver".driverData.pL1 < "InstE2MenergyMeterDriver".driverData.pL1Min OR "InstE2MenergyMeterDriver".driverData.pL1Min = 0.0 THEN
       "InstE2MenergyMeterDriver".driverData.pL1Min := "InstE2MenergyMeterDriver".driverData.pL1;
   END_IF;
   IF "InstE2MenergyMeterDriver".driverData.pL1 > "InstE2MenergyMeterDriver".driverData.pL1Max OR "InstE2MenergyMeterDriver".driverData.pL1Max = 0.0 THEN
       "InstE2MenergyMeterDriver".driverData.pL1Max := "InstE2MenergyMeterDriver".driverData.pL1;
   END_IF;

   IF "InstE2MenergyMeterDriver".driverData.pL2 < "InstE2MenergyMeterDriver".driverData.pL2Min OR "InstE2MenergyMeterDriver".driverData.pL2Min = 0.0 THEN
       "InstE2MenergyMeterDriver".driverData.pL2Min := "InstE2MenergyMeterDriver".driverData.pL2;
   END_IF;
   IF "InstE2MenergyMeterDriver".driverData.pL2 > "InstE2MenergyMeterDriver".driverData.pL2Max OR "InstE2MenergyMeterDriver".driverData.pL2Max = 0.0 THEN
       "InstE2MenergyMeterDriver".driverData.pL2Max := "InstE2MenergyMeterDriver".driverData.pL2;
   END_IF;

   IF "InstE2MenergyMeterDriver".driverData.pL3 < "InstE2MenergyMeterDriver".driverData.pL3Min OR "InstE2MenergyMeterDriver".driverData.pL3Min = 0.0 THEN
       "InstE2MenergyMeterDriver".driverData.pL3Min := "InstE2MenergyMeterDriver".driverData.pL3;
   END_IF;
   IF "InstE2MenergyMeterDriver".driverData.pL3 > "InstE2MenergyMeterDriver".driverData.pL3Max OR "InstE2MenergyMeterDriver".driverData.pL3Max = 0.0 THEN
       "InstE2MenergyMeterDriver".driverData.pL3Max := "InstE2MenergyMeterDriver".driverData.pL3;
   END_IF;

   IF "InstE2MenergyMeterDriver".driverData.pTotal < "InstE2MenergyMeterDriver".driverData.pTotalMin OR "InstE2MenergyMeterDriver".driverData.pTotalMin = 0.0 THEN
       "InstE2MenergyMeterDriver".driverData.pTotalMin := "InstE2MenergyMeterDriver".driverData.pTotal;
   END_IF;
   IF "InstE2MenergyMeterDriver".driverData.pTotal > "InstE2MenergyMeterDriver".driverData.pTotalMax OR "InstE2MenergyMeterDriver".driverData.pTotalMax = 0.0 THEN
       "InstE2MenergyMeterDriver".driverData.pTotalMax := "InstE2MenergyMeterDriver".driverData.pTotal;
   END_IF;

   // Reactive power
   "InstE2MenergyMeterDriver".driverData.qL1 := "Reactive power L1";
   "InstE2MenergyMeterDriver".driverData.qL2 := "Reactive power L2";
   "InstE2MenergyMeterDriver".driverData.qL3 := "Reactive power L3";
   "InstE2MenergyMeterDriver".driverData.qTotal := "PAC3220InPut"."Total_reactive_power_(VARn)";

   IF "InstE2MenergyMeterDriver".driverData.qL1 < "InstE2MenergyMeterDriver".driverData.qL1Min OR "InstE2MenergyMeterDriver".driverData.qL1Min = 0.0 THEN
       "InstE2MenergyMeterDriver".driverData.qL1Min := "InstE2MenergyMeterDriver".driverData.qL1;
   END_IF;
   IF "InstE2MenergyMeterDriver".driverData.qL1 > "InstE2MenergyMeterDriver".driverData.qL1Max OR "InstE2MenergyMeterDriver".driverData.qL1Max = 0.0 THEN
       "InstE2MenergyMeterDriver".driverData.qL1Max := "InstE2MenergyMeterDriver".driverData.qL1;
   END_IF;

   IF "InstE2MenergyMeterDriver".driverData.qL2 < "InstE2MenergyMeterDriver".driverData.qL2Min OR "InstE2MenergyMeterDriver".driverData.qL2Min = 0.0 THEN
       "InstE2MenergyMeterDriver".driverData.qL2Min := "InstE2MenergyMeterDriver".driverData.qL2;
   END_IF;
   IF "InstE2MenergyMeterDriver".driverData.qL2 > "InstE2MenergyMeterDriver".driverData.qL2Max OR "InstE2MenergyMeterDriver".driverData.qL2Max = 0.0 THEN
       "InstE2MenergyMeterDriver".driverData.qL2Max := "InstE2MenergyMeterDriver".driverData.qL2;
   END_IF;

   IF "InstE2MenergyMeterDriver".driverData.qL3 < "InstE2MenergyMeterDriver".driverData.qL3Min OR "InstE2MenergyMeterDriver".driverData.qL3Min = 0.0 THEN
       "InstE2MenergyMeterDriver".driverData.qL3Min := "InstE2MenergyMeterDriver".driverData.qL3;
   END_IF;
   IF "InstE2MenergyMeterDriver".driverData.qL3 > "InstE2MenergyMeterDriver".driverData.qL3Max OR "InstE2MenergyMeterDriver".driverData.qL3Max = 0.0 THEN
       "InstE2MenergyMeterDriver".driverData.qL3Max := "InstE2MenergyMeterDriver".driverData.qL3;
   END_IF;

   IF "InstE2MenergyMeterDriver".driverData.qTotal < "InstE2MenergyMeterDriver".driverData.qTotalMin OR "InstE2MenergyMeterDriver".driverData.qTotalMin = 0.0 THEN
       "InstE2MenergyMeterDriver".driverData.qTotalMin := "InstE2MenergyMeterDriver".driverData.qTotal;
   END_IF;
   IF "InstE2MenergyMeterDriver".driverData.qTotal > "InstE2MenergyMeterDriver".driverData.qTotalMax OR "InstE2MenergyMeterDriver".driverData.qTotalMax = 0.0 THEN
       "InstE2MenergyMeterDriver".driverData.qTotalMax := "InstE2MenergyMeterDriver".driverData.qTotal;
   END_IF;

   // Energy Tarif
   "InstE2MenergyMeterDriver".driverData.eActiveRate1Import := "Active energy import tariff 1(F)";
   "InstE2MenergyMeterDriver".driverData.eReactiveRate1Import := "Reactive energy import tariff 1 (F)";
   "InstE2MenergyMeterDriver".driverData.eApparentRate1Import := "Apparent energy tariff 1 (F)";
   "InstE2MenergyMeterDriver".driverData.eActiveRate1Export := "Active energy export tariff 1(F)";
   "InstE2MenergyMeterDriver".driverData.eReactiveRate1Export := "Reactive energy export tariff 1 (F)";






   // Reset 
   IF "InstEmDataHmi".statResetMinMaxAll  THEN

       // 모든 Min/Max 초기화 (Actual 값으로)
       "InstE2MenergyMeterDriver".driverData.uL1Min := 0.0;
       "InstE2MenergyMeterDriver".driverData.uL1Max := 0.0;
       "InstE2MenergyMeterDriver".driverData.uL2Min := 0.0;
       "InstE2MenergyMeterDriver".driverData.uL2Max := 0.0;
       "InstE2MenergyMeterDriver".driverData.uL3Min := 0.0;
       "InstE2MenergyMeterDriver".driverData.uL3Max := 0.0;

       "InstE2MenergyMeterDriver".driverData.uL1L2Min := 0.0;
       "InstE2MenergyMeterDriver".driverData.uL1L2Max := 0.0;
       "InstE2MenergyMeterDriver".driverData.uL2L3Min := 0.0;
       "InstE2MenergyMeterDriver".driverData.uL2L3Max := 0.0;
       "InstE2MenergyMeterDriver".driverData.uL3L1Min := 0.0;
       "InstE2MenergyMeterDriver".driverData.uL3L1Max := 0.0;

       "InstE2MenergyMeterDriver".driverData.uPhNaverageMin := 0.0;
       "InstE2MenergyMeterDriver".driverData.uPhNaverageMax := 0.0;

       "InstE2MenergyMeterDriver".driverData.uPhPhAverageMin := 0.0;
       "InstE2MenergyMeterDriver".driverData.uPhPhAverageMax := 0.0;

       "InstE2MenergyMeterDriver".driverData.iL1Min := 0.0;
       "InstE2MenergyMeterDriver".driverData.iL1Max := 0.0;
       "InstE2MenergyMeterDriver".driverData.iL2Min := 0.0;
       "InstE2MenergyMeterDriver".driverData.iL2Max := 0.0;
       "InstE2MenergyMeterDriver".driverData.iL3Min := 0.0;
       "InstE2MenergyMeterDriver".driverData.iL3Max := 0.0;

       "InstE2MenergyMeterDriver".driverData.iAverageMin := 0.0;
       "InstE2MenergyMeterDriver".driverData.iAverageMax := 0.0;

       "InstE2MenergyMeterDriver".driverData.cosL1Min := 0.0;
       "InstE2MenergyMeterDriver".driverData.cosL1Max := 0.0;
       "InstE2MenergyMeterDriver".driverData.cosL2Min := 0.0;
       "InstE2MenergyMeterDriver".driverData.cosL2Max := 0.0;
       "InstE2MenergyMeterDriver".driverData.cosL3Min := 0.0;
       "InstE2MenergyMeterDriver".driverData.cosL3Max := 0.0;

       "InstE2MenergyMeterDriver".driverData.cosAverageMin := 0.0;
       "InstE2MenergyMeterDriver".driverData.cosAverageMax := 0.0;

       "InstE2MenergyMeterDriver".driverData.fMin := 0.0;
       "InstE2MenergyMeterDriver".driverData.fMax := 0.0;

       "InstE2MenergyMeterDriver".driverData.pTotalMin := 0.0;
       "InstE2MenergyMeterDriver".driverData.pTotalMax := 0.0;
       "InstE2MenergyMeterDriver".driverData.qTotalMin := 0.0;
       "InstE2MenergyMeterDriver".driverData.qTotalMax := 0.0;
       "InstE2MenergyMeterDriver".driverData.sTotalMin := 0.0;
       "InstE2MenergyMeterDriver".driverData.sTotalMax := 0.0;

       "InstE2MenergyMeterDriver".driverData.sL1Min := 0.0;
       "InstE2MenergyMeterDriver".driverData.sL1Max := 0.0;
       "InstE2MenergyMeterDriver".driverData.sL2Min := 0.0;
       "InstE2MenergyMeterDriver".driverData.sL2Max := 0.0;
       "InstE2MenergyMeterDriver".driverData.sL3Min := 0.0;
       "InstE2MenergyMeterDriver".driverData.sL3Max := 0.0;

       "InstE2MenergyMeterDriver".driverData.pL1Min := 0.0;
       "InstE2MenergyMeterDriver".driverData.pL1Max := 0.0;
       "InstE2MenergyMeterDriver".driverData.pL2Min := 0.0;
       "InstE2MenergyMeterDriver".driverData.pL2Max := 0.0;
       "InstE2MenergyMeterDriver".driverData.pL3Min := 0.0;
       "InstE2MenergyMeterDriver".driverData.pL3Max := 0.0;

       "InstE2MenergyMeterDriver".driverData.qL1Min := 0.0;
       "InstE2MenergyMeterDriver".driverData.qL1Max := 0.0;
       "InstE2MenergyMeterDriver".driverData.qL2Min := 0.0;
       "InstE2MenergyMeterDriver".driverData.qL2Max := 0.0;
       "InstE2MenergyMeterDriver".driverData.qL3Min := 0.0;
       "InstE2MenergyMeterDriver".driverData.qL3Max := 0.0;

   END_IF;
END_REGION

REGION Network 4: Rangierung AI_EnergyMeter-Daten in HMI-Bereich / Routing AI_EnergyMeter data to HMI interface
   // Aufruf des FB Lsicar_EnMeterDataToHmi / Call of Lsicar_EnMeterDataToHmi FB
   RUNG wire#powerrail
      "InstEmDataHmi"(energyMeter01Visu := "InstE2MenergyMeterDriver".driverData, energyMeter02Visu :=, energyMeter03Visu :=, energyMeter04Visu :=, energyMeter05Visu :=, energyMeter06Visu :=, energyMeter07Visu :=, energyMeter08Visu :=)
   END_RUNG
   // the same network as SCL:
   "InstEmDataHmi"(energyMeter01Visu := "InstE2MenergyMeterDriver".driverData);   // "LSicar_EnMeterDataToHmi"
END_REGION
END_FUNCTION

FUNCTION "CallEnEffMonitor" : Void   // FC32, LAD
TITLE = CallEnergyEfficencyMonitor
AUTHOR : SICAR
FAMILY : Energy_EEM
VERSION : 1.0
// EEM  Verwaltung / The S7 Energy Efficiency-Monitor (or S7 EE-Monitor) allows you to record the energy consumption of your machine in a SIMATIC controller, and to analyze the results on the basis of the energy and media requirements.
// stored: IsIECCheckEnabled true, SetENOAutomatically true
   VAR_TEMP
      tempMeasPointIndex : USInt;   // HMI Index / HMI index
      tempCycleCounterAvgCalc : DInt;   // Umrechnung zu TOD / Calculation to TOD
      tempPlantInProduction : Bool;   // Anlage produziert / Plant in production
      tempReturnValue : Int;   // Temporary value for storing the EnPi reset time / Temporärer Wert zur Speicherung der EnPi-Resetzeit
   END_VAR
   // Ret_Val : Ret_Val
   VAR_TEMP   // added for the SCL form of the ladder/FBD networks
      _w1 : Bool;
      _w2 : Bool;
      _w3 : Bool;
      _w4 : Bool;
   END_VAR
BEGIN

REGION Network 1: Änderungshistorie / BLOCK INFO HEADER
   // Die Änderungshistorie wird nur in englischer Editiersprache geführt.
   // SIEMENS AG / (c)Copyright 2023
   // ------------------------------------------------------------------------------
   // Title:            CallEnEffMonitor (FC32)
   // Comment/Function: Call of Demo EnergyMeter and Energy Efficient M for EEMM demonstration
   // Library/Family:   Energy
   // Author:           SICAR
   // Tested with:      ---
   // Engineering:      TIA Portal V19
   // Restrictions:     -
   // Requirements:     ---
   // ------------------------------------------------------------------------------
   // Change log table:
   // Version  | Date       | Expert in charge       | Changes applied
   // ---------|------------|------------------------|------------------------------
   // 05.00.00 | 01.09.2023 | SICAR
   //                         First released version
END_REGION

REGION Network 2: DESCRIPTION
   // The Energy Efficiency Monitor “EEM” integrated in SICAR is based on the application example in entry ID: 109753230 V1.0 dated 02/2018 of the Siemens Industry Online Support, see: 
   // 
   // https://support.industry.siemens.com/cs/document/109753230/-s7-energy-efficiency-monitor-for-machines?dti=0&lc=en-WW 
   // 
   // **License**  
   // The software package has to be licensed. The necessary license key has to be entered in the data block for energy data “EEmData”, in the array item “licenseKey”. 
   //  
   // {.pageWidth}
   // ![Image](EemEnPiCalc/en/image1.PNG)
   // 
   // The S7 Energy Efficiency-Monitor (or S7 EE-Monitor) allows you to record the energy consumption of your machine in a SIMATIC controller, and to analyze the results on the basis of the energy and media requirements.  
   // https://support.industry.siemens.com/cs/document/109753230/s7-energieeffizienz-monitor-für-maschinen?dti=0&lc=de-WW 
   // 
   // **PLC Data types**  
   //  LSicar_typeEeMenPiCalc 
   //  LSicar_typeEeMenPiEstate 
   //  LSicar_typeEeMenPiLimit 
   //  typeEnMeterOutputData 
   //  typeMeasDataProfileE3 
   //  
   // **WinCC Faceplates**  
   // 
   // ![Image](EemEnPiCalc/en/image3.PNG)
   // 
   // **WinCC Screen**  
   //  
   // ![Image](EemEnPiCalc/en/image4.PNG)
   //  
   // # Devices & networks 
   // 
   // An additional AI Energy Meter has been added and configured in the SICAR project. The user data has been  
   // configured as module version “EE@Industry measured data profile e3”.  
   // 
   // Select the module version according to your requirements. The data assignment in the FC blocks has to be adjusted according to the selected module version. 
   // 
   // ![Image](EemEnPiCalc/en/image5.PNG)
   //  
   //  
   // 
   //  #### PLC Programm blocks 
   // 
   // ##### CallEnSeem  
   // The block is called in OB “CYCLIC_INTERRUPT_100MS_OB” (100ms cycle). The block contains the following instructions which can be found in “Instructions > Optional packages > Energy Suite extensions”.
   // 
   // **EnS_EEm_Calc:**  
   // The instruction calculates operating state-related energy data of machines and plants for uniform efficiency evaluation, in accordance with the VDMA 34179 measuring directive. 
   // 
   // ---
   // Note
   // :     The instruction calculates the energy efficiency value of the respective state for up to 8 operating states, and the global energy efficiency value. 
   // :     The maximum number of configurable measuring points is 10. Refer to the documentation of the entry ID. 
   // 
   // ---
   // 
   // **EnS_EEm_Report:**  
   // The instruction writes the data for the efficiency report to the data log on the SIMATIC memory card, in accordance with the VDMA 34179 measuring directive. The data log is a CSV file. 
   // 
   // ##### CallEnEffMonitor
   // ---
   // Note
   // :     The assignment of the readings as well as the formation of additional signals can be represented only exemplarily here. It has to be adapted to the actual plant conditions! 
   // 
   // ---
   // 
   // * Networks 1 & 2: The readings of the two AI-Energy-Meters are entered in the DB “EeMonitor”, in an array [0..9] in accordance with the measurement data profile “typeMeasDataProfileE3”. 
   // * Network 3: According to the selection of a measuring point on the HMI, data of the respective measuring point is routed to the HMI data area. The selection is done with a Pull-Down menu and a symbolic I/O field. 
   // * Network 4: Several tags in the EnS…data types are not marked as accessible / visible. In order to display these tags on the HMI all the same, they are routed to DB “EeMonitor” in structure “typeEnMeterWorkHmi”. There the tags are marked as accessible / visible.  
   // * Network 5: A collective signal is generated, according to the exemplary calls for OP area 1. This is only an example! The collective signal shows that the plant is producing parts, by a disjunction (OR) of all outputs. If an output is controlled, the plant is moving and producing parts. This collective signal is used later on to generate the energetic states “eState”. A delay of 3 seconds has been configured so that a short break in controlling the outputs will not change the energetic state. *
   // * Network 6: The signals for the energetic states are generated here. 
   // * Network 7: Simulation On/Off: A part counter is simulated here. Note: the simulation can be switched on and off with a button in the screen. 
   // * Network 8: Simulation On/Off. Energy counters for both AI-Energy-Meters are simulated here. Note: the simulation can be switched on and off with a button in the screen. 
   // * Network 9: Call of blocks “EemDemoSimulation” and “EemDemoResetValEMeter”. 
   // * Network 10: Call of block “EemEnPiCalc” and data routing according to the selection of a measuring point on the HMI. 
   // * Network 11: Error evaluation of block “EemEnPiCalc” to generate ProDiag messages. 
   // * Network 12: Error evaluation of block “EnS_EEm_Report” to generate ProDiag messages.  
   // 
   // ##### EemDemoResetValEMeter  
   // 
   // The block resets certain measurement values by controlling the respective outputs in the I/O area of the AI-Energy-Meter. 
   // 
   // ##### EemDemoSimulation  
   // 
   // This block simulates higher or lower energy values, according to the energetic states “eState”. 
   // 
   // ##### EemEnPiCalc
   // This block calculates the ENPI (Energy value Pro Item). It substitutes the script “EEm_EnPI_Efficiency” of the entry ID. 
   // 
   // ---
   // Note
   // :     All block parameters are provided with “pre-defined actual parameters”.
   // 
   // ---
   // 
   // **Operation mode Automatic / Manual**  
   // 
   // The blocks are independent of operation modes. Therefor they are not assigned to any operation mode area. 
   // 
   // **PLC Alarm text list**  
   // 
   // The following PLC alarm text lists have been created: 
   // 
   // * **EEMonitor_Calc_Warn_PD** ProDiag alarm text list for alarms by instruction “EnS_EEm_Calc”.   
   // * **EEMonitor_Report_Warn_PD** ProDiag alarm text list for alarms by instruction “EnS_EEm_Report”.   
   // Both PLC alarm text lists have been entered in the PLC alarm text list “GLOBAL_GENERAL_AlarmTextList”. 
   // 
   // ---
   // Note
   // :     The alarm texts are provided in two languages (German, English). Please consider the multilingual nature of the entries. 
   // 
   // ---
   // 
   // #### PLC Data types 
   // 
   // PLC data types used for PLC program block or HMI faceplate:  
   // ![Image](_Icon/reference.PNG)  See ..\Library Types\LSicar_typeEeMenPiCalc.pdf  
   // 
   // #### WinCC Objects 
   // 
   // **WinCC HMI-tags**  
   // 
   // The HMI tags are stored in the tag table “AI_EnergyMeter_EEM” in the SICAR project.  
   // 
   // **WinCC Text and graphics lists**  
   // 
   // The text list “EE-MONITOR_MEASUREPOINT” contains the texts necessary for the pull-down menu / symbolic I/O field in the screen. Please take into account the multilingual nature of the entries.  
   // 
   // **WinCC Faceplates**  
   // 
   // The faceplates are stored in the project library, in folder “types”. They have been created using several WinCC objects; they are animated depending on the state. 
   // 
   // * EEM_EnPI_EnergyPerItem:	display of ENPI (ENergy Per Item) 
   // * EEM_ViewBar_Diff-AVG-REF:	bar display to compare reference value and average value 
   // * EEM_ViewBar_EState-Total:	bar display of energy status (not used at this time) 
   // * EEM_ViewBarCurve_EState:	Total: bar display and curve display of the energy values  
   // 
   // **WinCC-screen** 
   // 
   // 1. HMI Screens:	EE-MONITOR_ENERGY: display of the energy values 
   // 2. HMI Popup-screens 
   // 	* EEM_LEGEND_Popup: 		Legend 
   // 	* EEM_INFO-MACHINE_Popup: 	Machine information 
   // 	* EEM_STARTMEASURE_Popup: 	Popup to start the normal measurement or the reference measurement  
   // 	* EEM_UIPE_Popup: 		display of voltage, current, power, and energy 
   // 	* MORE_EEM_Popup: 		Popup with additional buttons 
   // 	* MORE_AddOn_Popup: 		supplemented  with button “EE-Monitor” 
   // 
   //  
   // 
   // {.pageWidth}
   // ![Image](EemEnPiCalc/en/image6.PNG)
   //  
   //  
   // 
   // #### Additional information
   // 
   // #### Update info
   // 
   // #### Further documentations
END_REGION

REGION Network 3: select measurement values
   // can be from EnergyMeter driver or directly from any hardware (in this example EnergyMeter module and PAC)
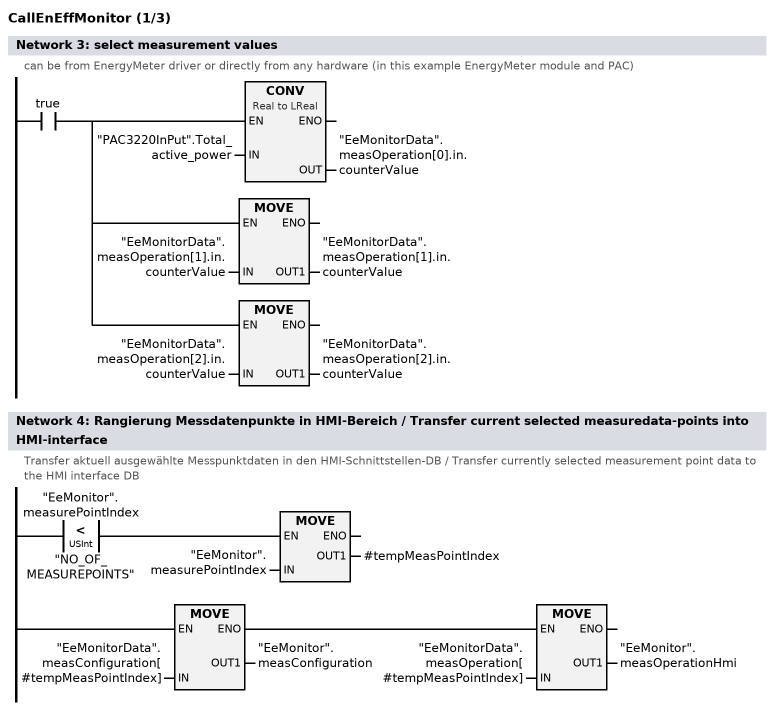
   RUNG wire#powerrail
      Contact( true )
      wire#w1
      { S7_Templates := "[SrcType := Real, DestType := LReal]" } Convert(in := "PAC3220InPut".Total_active_power, out => "EeMonitorData".measOperation[0].in.counterValue)
   END_RUNG
   RUNG wire#w1
      Move(in := "EeMonitorData".measOperation[1].in.counterValue, out1 => "EeMonitorData".measOperation[1].in.counterValue)
   END_RUNG
   RUNG wire#w1
      Move(in := "EeMonitorData".measOperation[2].in.counterValue, out1 => "EeMonitorData".measOperation[2].in.counterValue)
   END_RUNG
   // the same network as SCL:
   IF true THEN
       "EeMonitorData".measOperation[0].in.counterValue := REAL_TO_LREAL("PAC3220InPut".Total_active_power);
       "EeMonitorData".measOperation[1].in.counterValue := "EeMonitorData".measOperation[1].in.counterValue;
       "EeMonitorData".measOperation[2].in.counterValue := "EeMonitorData".measOperation[2].in.counterValue;
   END_IF;
END_REGION

REGION Network 4: Rangierung Messdatenpunkte in HMI-Bereich / Transfer current selected measuredata-points into HMI-interface
   // Transfer aktuell ausgewählte Messpunktdaten in den HMI-Schnittstellen-DB / Transfer currently selected measurement point data to the HMI interface DB
   RUNG wire#powerrail
      { S7_Templates := "SrcType := USInt" } LT_Contact(in1 := "EeMonitor".measurePointIndex, in2 := "NO_OF_MEASUREPOINTS")
      Move(in := "EeMonitor".measurePointIndex, out1 => #tempMeasPointIndex)
   END_RUNG
   RUNG wire#powerrail
      Move(in := "EeMonitorData".measConfiguration[#tempMeasPointIndex], out1 => "EeMonitor".measConfiguration)
      Move(in := "EeMonitorData".measOperation[#tempMeasPointIndex], out1 => "EeMonitor".measOperationHmi)
   END_RUNG
   // the same network as SCL:
   IF "EeMonitor".measurePointIndex < "NO_OF_MEASUREPOINTS" THEN
       #tempMeasPointIndex := "EeMonitor".measurePointIndex;
   END_IF;
   "EeMonitor".measConfiguration := "EeMonitorData".measConfiguration[#tempMeasPointIndex];
   "EeMonitor".measOperationHmi := "EeMonitorData".measOperation[#tempMeasPointIndex];
END_REGION

REGION Network 5: WORKaround: Rangierung / WORKaround: Transfer data from EeMonitroData to EeMonitor.work
   // Konvertierung Zeit in DTL und addieren Zeitzone mit Datum und Uhrzeit aus EnS_EEm_Calc zur Darstellung des tatsächlichen Datums und der tatsächlichen Uhrzeit im aktuellen Land.
   // Convertion of Time to DTL and adding time zone with date and time taken from EnS_EEm_Calc for representing the actual date and time in the current country.
   // Data is copied from EeMonitorData to EeMonitor.work
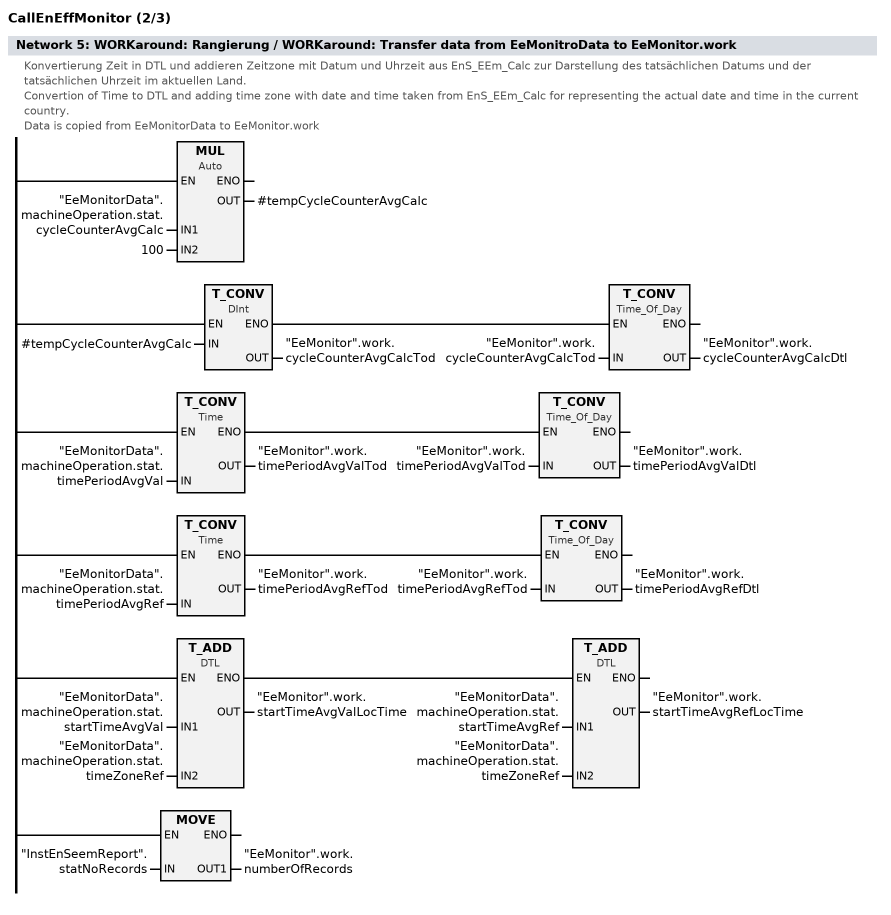
   RUNG wire#powerrail
      Mul(in1 := "EeMonitorData".machineOperation.stat.cycleCounterAvgCalc, in2 := 100, out => #tempCycleCounterAvgCalc)
   END_RUNG
   RUNG wire#powerrail
      { S7_Templates := "[src_type := DInt, dest_type := Time_Of_Day]" } T_CONV(IN := #tempCycleCounterAvgCalc, OUT => "EeMonitor".work.cycleCounterAvgCalcTod)
      { S7_Templates := "[src_type := Time_Of_Day, dest_type := DTL]" } T_CONV(IN := "EeMonitor".work.cycleCounterAvgCalcTod, OUT => "EeMonitor".work.cycleCounterAvgCalcDtl)
   END_RUNG
   RUNG wire#powerrail
      { S7_Templates := "[src_type := Time, dest_type := Time_Of_Day]" } T_CONV(IN := "EeMonitorData".machineOperation.stat.timePeriodAvgVal, OUT => "EeMonitor".work.timePeriodAvgValTod)
      { S7_Templates := "[src_type := Time_Of_Day, dest_type := DTL]" } T_CONV(IN := "EeMonitor".work.timePeriodAvgValTod, OUT => "EeMonitor".work.timePeriodAvgValDtl)
   END_RUNG
   RUNG wire#powerrail
      { S7_Templates := "[src_type := Time, dest_type := Time_Of_Day]" } T_CONV(IN := "EeMonitorData".machineOperation.stat.timePeriodAvgRef, OUT => "EeMonitor".work.timePeriodAvgRefTod)
      { S7_Templates := "[src_type := Time_Of_Day, dest_type := DTL]" } T_CONV(IN := "EeMonitor".work.timePeriodAvgRefTod, OUT => "EeMonitor".work.timePeriodAvgRefDtl)
   END_RUNG
   RUNG wire#powerrail
      { S7_Templates := "[date_type := DTL, time_type := Time]" } T_ADD(IN1 := "EeMonitorData".machineOperation.stat.startTimeAvgVal, IN2 := "EeMonitorData".machineOperation.stat.timeZoneRef, OUT => "EeMonitor".work.startTimeAvgValLocTime)
      { S7_Templates := "[date_type := DTL, time_type := Time]" } T_ADD(IN1 := "EeMonitorData".machineOperation.stat.startTimeAvgRef, IN2 := "EeMonitorData".machineOperation.stat.timeZoneRef, OUT => "EeMonitor".work.startTimeAvgRefLocTime)
   END_RUNG
   RUNG wire#powerrail
      Move(in := "InstEnSeemReport".statNoRecords, out1 => "EeMonitor".work.numberOfRecords)
   END_RUNG
   // the same network as SCL:
   #tempCycleCounterAvgCalc := "EeMonitorData".machineOperation.stat.cycleCounterAvgCalc * 100;
   T_CONV(IN := #tempCycleCounterAvgCalc, OUT => "EeMonitor".work.cycleCounterAvgCalcTod, ENO => #_w1);
   IF #_w1 THEN
       T_CONV(IN := "EeMonitor".work.cycleCounterAvgCalcTod, OUT => "EeMonitor".work.cycleCounterAvgCalcDtl);
   END_IF;
   T_CONV(IN := "EeMonitorData".machineOperation.stat.timePeriodAvgVal,
          OUT => "EeMonitor".work.timePeriodAvgValTod,
          ENO => #_w2);
   IF #_w2 THEN
       T_CONV(IN := "EeMonitor".work.timePeriodAvgValTod, OUT => "EeMonitor".work.timePeriodAvgValDtl);
   END_IF;
   T_CONV(IN := "EeMonitorData".machineOperation.stat.timePeriodAvgRef,
          OUT => "EeMonitor".work.timePeriodAvgRefTod,
          ENO => #_w3);
   IF #_w3 THEN
       T_CONV(IN := "EeMonitor".work.timePeriodAvgRefTod, OUT => "EeMonitor".work.timePeriodAvgRefDtl);
   END_IF;
   T_ADD(IN1 := "EeMonitorData".machineOperation.stat.startTimeAvgVal,
         IN2 := "EeMonitorData".machineOperation.stat.timeZoneRef,
         OUT => "EeMonitor".work.startTimeAvgValLocTime,
         ENO => #_w4);
   IF #_w4 THEN
       T_ADD(IN1 := "EeMonitorData".machineOperation.stat.startTimeAvgRef,
             IN2 := "EeMonitorData".machineOperation.stat.timeZoneRef,
             OUT => "EeMonitor".work.startTimeAvgRefLocTime);
   END_IF;
   "EeMonitor".work.numberOfRecords := "InstEnSeemReport".statNoRecords;
END_REGION

REGION Network 6: Betriebsarten für BA-Bereich1 auf "eState" in "EEm_Data_DB" / Operation modes to "eState"
   // Setzt Estate Nummer abhängig vom ausgewählten OpMode1-Modus / Sets Estate number accoriding to the selected state
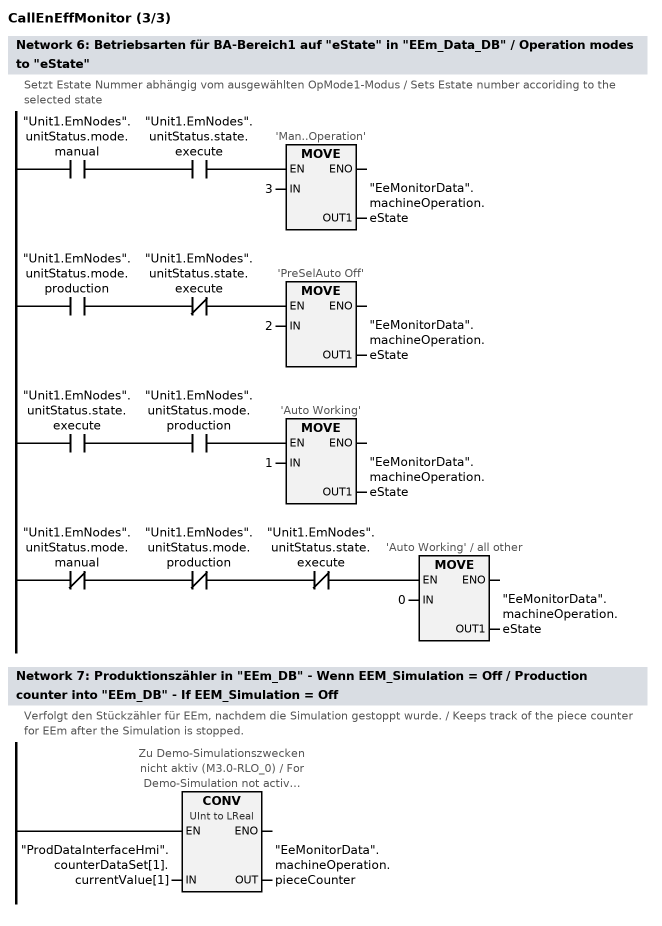
   RUNG wire#powerrail
      Contact( "Unit1.EmNodes".unitStatus.mode.manual )
      Contact( "Unit1.EmNodes".unitStatus.state.execute )
      Move(in := 3, out1 => "EeMonitorData".machineOperation.eState)   // 'Man..Operation'
   END_RUNG
   RUNG wire#powerrail
      Contact( "Unit1.EmNodes".unitStatus.mode.production )
      I_Contact( "Unit1.EmNodes".unitStatus.state.execute )
      Move(in := 2, out1 => "EeMonitorData".machineOperation.eState)   // 'PreSelAuto Off'
   END_RUNG
   RUNG wire#powerrail
      Contact( "Unit1.EmNodes".unitStatus.state.execute )
      Contact( "Unit1.EmNodes".unitStatus.mode.production )
      Move(in := 1, out1 => "EeMonitorData".machineOperation.eState)   // 'Auto Working'
   END_RUNG
   RUNG wire#powerrail
      I_Contact( "Unit1.EmNodes".unitStatus.mode.manual )
      I_Contact( "Unit1.EmNodes".unitStatus.mode.production )
      I_Contact( "Unit1.EmNodes".unitStatus.state.execute )
      Move(in := 0, out1 => "EeMonitorData".machineOperation.eState)   // 'Auto Working' / all other
   END_RUNG
   // the same network as SCL:
   IF "Unit1.EmNodes".unitStatus.mode.manual AND "Unit1.EmNodes".unitStatus.state.execute THEN
       "EeMonitorData".machineOperation.eState := 3;   // 'Man..Operation'
   END_IF;
   IF "Unit1.EmNodes".unitStatus.mode.production AND NOT "Unit1.EmNodes".unitStatus.state.execute THEN
       "EeMonitorData".machineOperation.eState := 2;   // 'PreSelAuto Off'
   END_IF;
   IF "Unit1.EmNodes".unitStatus.state.execute AND "Unit1.EmNodes".unitStatus.mode.production THEN
       "EeMonitorData".machineOperation.eState := 1;   // 'Auto Working'
   END_IF;
   IF NOT "Unit1.EmNodes".unitStatus.mode.manual AND NOT "Unit1.EmNodes".unitStatus.mode.production AND NOT "Unit1.EmNodes".unitStatus.state.execute THEN
       "EeMonitorData".machineOperation.eState := 0;   // 'Auto Working' / all other
   END_IF;
END_REGION

REGION Network 7: Produktionszähler in "EEm_DB" - Wenn EEM_Simulation = Off / Production counter into "EEm_DB" - If EEM_Simulation = Off
   // Verfolgt den Stückzähler für EEm, nachdem die Simulation gestoppt wurde. / Keeps track of the piece counter for EEm after the Simulation is stopped.
   RUNG wire#powerrail
      { S7_Templates := "[SrcType := UInt, DestType := LReal]" } Convert(in := "ProdDataInterfaceHmi".counterDataSet[1].currentValue[1], out => "EeMonitorData".machineOperation.pieceCounter)   // Zu Demo-Simulationszwecken nicht aktiv (M3.0-RLO_0) / For Demo-Simulation not active (M3.0-RLO_0)
   END_RUNG
   // the same network as SCL:
   "EeMonitorData".machineOperation.pieceCounter := UINT_TO_LREAL("ProdDataInterfaceHmi".counterDataSet[1].currentValue[1]);   // Zu Demo-Simulationszwecken nicht aktiv (M3.0-RLO_0) / For Demo-Simulation not active (M3.0-RLO_0)
END_REGION

REGION Network 8 (SCL): Temporary value for storing the EnPi reset time / Reset EnPI values
   // Liest die aktuelle Uhrzeit und speichert sie, um dem Benutzer Informationen über den letzten EnPi-Reset bereitzustellen / Reads the current time and store it to provide the user the information about the last EnPi reset
   // Check for the trigger to reset/recalculate the EnPI values
   IF ("EeMonitorData".internalData.enpiResetTrigger = TRUE) THEN

       // Read the current time and store it to provide the user the information
       // about the last reset
       #tempReturnValue := RD_LOC_T("EeMonitorData".internalData.enpiResetTime);

       // Reset the trigger
       "EeMonitorData".internalData.enpiResetTrigger := FALSE;
   ELSE
       ; // No trigger
   END_IF;
END_REGION
END_FUNCTION

ORGANIZATION_BLOCK "Interrupt1s"   // OB31, LAD, CyclicInterrupt
TITLE = Zyklischer Interrupt 100ms / Cyclic interrupt 100ms
AUTHOR : SICAR
FAMILY : OB
VERSION : 1.0
// organisation block
// stored: IsIECCheckEnabled true, SetENOAutomatically true
   VAR_INPUT
      Initial_Call : Bool;   // Initial call of this OB
      Event_Count : Int;   // Events discarded
   END_VAR
BEGIN

REGION Network 1: Änderungshistorie / ChangeLog
   // Die Änderungshistorie wird nur in englischer Editiersprache geführt.
   // Change log table:
   // Version | Date | Expert in charge | Changes applied
   // -------|---------|-------------|--------------------------------------------
   // 01.00.00 | 01.01.1999 | Person x | First released version
   // 01.00.01 | 02.01.1999 | Person y | Block was Updated
END_REGION

REGION Network 2: EE-MONITOR: Aufruf & Mess-Daten in "EEmData_DB" / Call & measure-data into "EEmData_DB"
   // Aufruf der Energieeffizienz Überwachungs Functionen / Call the energy efficiency monitor functions
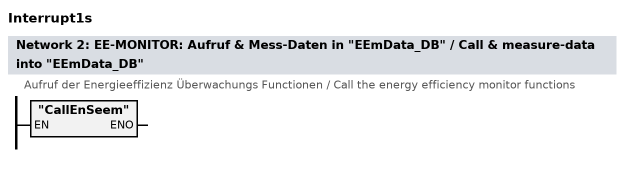
   RUNG wire#powerrail
      "CallEnSeem"()
   END_RUNG
   // the same network as SCL:
   "CallEnSeem"();
END_REGION
END_ORGANIZATION_BLOCK

FUNCTION "CallEnSeem" : Void   // FC34, LAD
TITLE = CallEnSeem
AUTHOR : SICAR
FAMILY : Energy_EEM
VERSION : 1.0
// Der in SICAR eingebaute Energie Effizienz Monitor „EEM“ basiert auf der Beitrags-ID: 109753230, V1.0 von 02/2018 des Siemens Industry Online Support, siehe:  
// https://support.industry.siemens.com/cs/document/109753230/s7-energieeffizienz-monitor-f%C3%BCr-maschinen?dti=0&lc=de-WW  
// 
// **Lizenz**  
// Das Softwarepaket ist Lizenzpflichtig. Die notwendige Lizenz muss im Datenbaustein der Energiedaten „EeMonitorData“ im Datum „licencsKey“ eingetragen werden.  
// 
// 
// Mit dem S7 Energieeffizienz-Monitor können Sie Energieverbräuche Ihrer Maschine in einer SIMATIC Steuerung erfassen und anhand des Energie- und Medienbedarfs statusbezogen anhand der energetischen Zustände analy-sieren. 
//  
//  
// **SPS-Programmbausteine**  
//  
// **PLC-Datentypen**  
//   LSicar_typeEeMenPiCalc  
//   LSicar_typeEeMenPiEstate  
//   LSicar_typeEeMenPiLimit  
//   typeEnMeterOutputData  
//   typeMeasDataProfileE3  
// 
// **WinCC-Bildbaustein**  
//  
// **WinCC-Bild**  
//  
//  
// #### Geräte & Netze
// Im SICAR-Projekt ist ein weiteres AI Energy Meter eingefügt und konfiguriert. Dies ist unter „Nutzdaten“ mit der Modulversion „EE@Industry Messdatenprofil e3“ parametriert.  
// Wählen Sie entsprechend Ihren Anforderungen die Modulversion aus. Je nach gewählter Modulversion, muss die Datenrangierung in den FC-Bausteinen angepasst werden.  
//  
// 
// #### SPS-Programmbausteine
// **CallEnSeem**  
// Der Baustein wird im OB „CYCLIC_INTERRUPT_100MS_OB“ (100ms Takt) aufgerufen. Darin sind nachfolgende Baustein-Anweisungen. Sie sind enthalten unter „Optionspakete > Energy Suite Erweiterungen“.  
// 
// **EnS_EEm_Calc:**  
// Der Baustein berechnet betriebszustandsbezogene Energiedaten von Maschinen und Anlagen zur einheitlichen Effizienzbewertung gemäß Messvorschrift VDMA 34179.  
// 
// NOTE
//  
// :     Der Baustein berechnet für bis zu acht Betriebszustände den Energieeffizienzwert des jeweiligen Zustands sowie den Gesamt-Energieeffizienzwert. 
// :     Die maximale Anzahl der konfigurierbaren Messstellen ist 10. Beachten Sie hierzu die Dokumentation der Beitrags-ID.
// 
// ---
// 
// **EnS_EEm_Report:**  
// Der Baustein erstellt ein Effizienzprotokoll im CSV-Format auf der SIMATIC Memory Card der CPU gemäß Messvorschrift VDMA 34179.  
// 
// **CallEnEffMonitor**  
// 
// NOTE
// :     Die Rangierung der Messdaten, sowie die Bildung von zusätzlichen Signalen kann hier nur beispiel-haft dargestellt werden. Sie muss auf die tatsächlichen Anlagengegebenheiten angepasst werden!
// 
// ---
// 
// * **Netzwerk 1 & 2:** In den beiden Netzwerken werden die Messdaten der beiden AI-Energy-Meter in den DB „EeMonitor“ einge-tragen, in ein Arrayfeld [0..9] gemäß dem Messdatenprofil " typeMeasDataProfileE3".
// * **Netzwerk 3:** Entsprechend des auf dem HMI angewählten Messpunktes (Pull-Down-Menü / Symbolisches E/A-Feld) wer-den hier die Daten des jeweiligen Messpunktes in dem HMI-Datenbereich rangiert.
// * **Netzwerk 4:** Einige Daten in den EnS…-Datentypen (im DB „EeMonitorData“) sind nicht mit Erreichbar/Sichtbar gekenn-zeichnet. Um diese Daten dennoch auf dem HMI darzustellen, werden sie in dem DB „EeMonitor“ rangiert in die Struktur „typeEnMeterWorkHmi“; dort sind die Daten mit Erreichbar/Sichtbar gekennzeichnet. 
// * **Netzwerk 5:** Hier wird ein Summensignal gebildet, entsprechend den Beispiel-Aufrufen für Betriebsartenbereich 1. Es han-delt sich hierbei lediglich um eine Beispiel-Anwendung! Das Summensignal gibt an, das die Anlage Teile pro-duziert. Hierzu werden alle Ausgänge verodert: Werden die Ausgänge angesteuert, so bewegt sich die Anla-ge, die Anlage produziert. Dieses Summensignal wird später benötigt, um damit die energetischen Zustände „eState“ zu bilden. Damit eine kurze Pause bzgl. der Ansteuerung der Ausgänge nicht zu einem Wechsel des energetischen Zustands führt ist hier eine Zeitverzögerung von 3 Sekunden eingebaut.
// * **Netzwerk 6:** In diesem Netzwerk werden die Signale für die energetischen Zustände gebildet.
// * **Netzwerk 7:** Simulation Ein/Aus Betrifft die Simulation von einem Stückzähler. Es wird hier ein simulierter Zähler als Stückzähler verwendet. Hinweis: Die Simulation kann im Bild mittels eines Buttons ein- und ausgeschaltet werden.
// * **Netzwerk 8:** Simulation Ein/Aus Betrifft die Simulation von Energiezähler für beide AI-Energy-Meter. Hinweis: Die Simulation kann im Bild mittels eines Button Ein- und Ausgeschaltet werden.
// * **Netzwerk 9:** Aufruf der Bausteine „EemDemoSimulation“ und „“EemDemoResetValEmeter“.
// * **Netzwerk 10:** Aufruf des Bausteins „EemEnPiCalc“ und Rangierung der daten entspr. dem auf dem HMI ausgewählten Messpunktes.
// * **Netzwerk 11:** Fehlerauswertung des Bausteins “ EemEnPiCalc“ zur Generierung von ProDiag-Meldungen.
// * **Netzwerk 12:** Fehlerauswertung des Bausteins “EnS_EEm_Report“ zur Generierung von ProDiag-Meldungen.
// 
// **EemDemoResetValEmeter** Der Baustein führt ein Reset auf gewisse Messwerte aus, durch Zuweisen der entspr. Ausgänge im E/A-Bereich der AI-Energy-Meter.
// **EemDemoSimulation** Baustein zur Simulation von höheren oder niedrigeren Energiewerten entsprechend der energetischen Zustände „eState“.
// **EemEnPiCalc** Der Baustein berechnet den ENPI (Energiewert Pro Item). Er ersetzt das Skript „EEm_EnPI_Efficiency“ der Bei-trags-ID.
// 
// **Parameter**  
// 
// NOTE
// :     Alle Bausteinparameter sind mit "Vordefinierten Aktualparametern" versehen.
// 
// ---
// 
// **Betriebsart Automatik / Hand** 
// Die Bausteine sind keinem Betriebsartenbereich zugeordnet.  
// 
// **PLC-Meldetextliste**  
// Folgende PLC-Meldetextlisten wurden hierzu angelegt:  
// * EEMonitor_Calc_Warn_PD Beinhaltet die ProDiag-Meldetext für den Bausteinaufruf „EnS_EEm_Calc“.  
// * EEMonitor_Report_Warn_PD Beinhaltet die ProDiag-Meldetexte für den Bausteinaufruf „EnS_EEm_Report“  
// 
// Beide Meldetextlisten sind in der PLC-Meldetextliste „GLOBAL_GENERAL_AlarmTextList“ eingetragen.  
// 
// NOTE
// :    Die Textlisten sind in Deutsch und Englisch ausgeführt. Bitte beachten Sie die Mehrsprachigkeit der PLC-Meldetextlisten.
// 
// ---
// 
// #### PLC-Datentypen
// Verwendete PLC-Datentypen für den SPS-Programmbaustein / WinCC-Bildbaustein:  
// Siehe ..\Library Types\LSicar_typeEeMenPiCalc.pdf  
//  
// #### WinCC-Objekte
// **WinCC HMI-Variablen**  
// Die HMI-Variablen sind im SICAR-Projekt angelegt in der Variablentabelle „AI_EnergyMeter_EEM“  
// 
// **WinCC Text- und Grafiklisten**  
// Die für das im Bild befindliche Pull-Down-Menü / Symbolisches E/A-Feld notwendigen Texte sind in der Text- und Grafikliste „EE-MONITOR_MEASUREPOINT“ hinterlegt. Bitte beachten Sie auch hier die Mehrsprachigkeit.  
// 
// **WinCC-Bildbaustein**  
// Die Bildbausteine befinden sich in der Projekt-Bibliothek unter „Typen“. Sie sind erstellt aus mehreren einzelnen WinCC-Objekten und animiert, je nach Zustand.  
// * EEM_EnPI_EnergyPerItem: Darstellung ENPI (Energy Per Item)
// * EEM_ViewBar_Diff-AVG-REF: Balkendarstellung zum Vergleich zwischen Referenz- / Durchschnittswert
// * EEM_ViewBar_EState-Total: Balkendarstellung Energie Status (z.Zt. nicht verwendet)
// * EEM_ViewBarCurve_EState-Total: Balken- und Kurvendarstellung der Energiewerte
// 
// **WinCC-Bild**  
// * HMI Bilder	
// 	- EE-MONITOR_ENERGY: Darstellung der Energiewerte
// * HMI Popup-Bilder	
// 	- EEM_LEGEND_Popup: Legende
// 	- EEM_INFO-MACHINE_Popup: Maschineninformationen
// 	- EEM_STARTMEASURE_Popup: Popup zum Starten der Normal- oder Referenzmessung
// 	- EEM_UIPE_Popup: Darstellung von Spannung, Strom, Leistung und Energie
// 	- MORE_EEM_Popup: Popup mit zusätzlichen Schaltflächen / Buttons
// 	- MORE_AddOn_Popup: Ergänzt um Button „EE-Monitor“
//  
// #### Weitere Hinweise
// 
// #### Updateinfo
// 
// #### Weitere Dokumente
// The S7 Energy Efficiency-Monitor (or S7 EE-Monitor) allows you to record the energy consumption of your machine in a SIMATIC controller, and to analyze the results on the basis of the energy and media requirements.
// stored: IsIECCheckEnabled true, SetENOAutomatically true
   // Ret_Val : Ret_Val
BEGIN

REGION Network 1: Änderungshistorie / BLOCK INFO HEADER
   // Die Änderungshistorie wird nur in englischer Editiersprache geführt.
   // SIEMENS AG / (c)Copyright 2023
   // ------------------------------------------------------------------------------
   // Title:            CallEnSeem (FC34)
   // Comment/Function: The S7 Energy Efficiency-Monitor (or S7 EE-Monitor) allows you to record the energy consumption of your machine in a SIMATIC controller, and to analyze the results on the basis of the energy and media requirements.
   // Library/Family:   Energy_EEM
   // Author:           SICAR
   // Tested with:      ---
   // Engineering:      TIA Portal V19
   // Restrictions:     -
   // Requirements:     ---
   // ------------------------------------------------------------------------------
   // Change log table:
   // Version | Date | Expert in charge | Changes applied
   // -------|---------|-------------|--------------------------------------------
   // 01.00.00 | 01.01.1999 | Person x | First released version
   // 01.00.01 | 02.01.1999 | Person y | Block was Updated
END_REGION

REGION Network 2: DESCRIPTION
   // The Energy Efficiency Monitor “EEM” integrated in SICAR is based on the application example in entry ID: 109753230 V1.0 dated 02/2018 of the Siemens Industry Online Support, see: 
   // 
   // https://support.industry.siemens.com/cs/document/109753230/-s7-energy-efficiency-monitor-for-machines?dti=0&lc=en-WW 
   // 
   // **License**  
   // The software package has to be licensed. The necessary license key has to be entered in the data block for energy data “EEmData”, in the array item “licenseKey”. 
   //  
   // {.pageWidth}
   // ![Image](EemEnPiCalc/en/image1.PNG)
   // 
   // The S7 Energy Efficiency-Monitor (or S7 EE-Monitor) allows you to record the energy consumption of your machine in a SIMATIC controller, and to analyze the results on the basis of the energy and media requirements.  
   // https://support.industry.siemens.com/cs/document/109753230/s7-energieeffizienz-monitor-für-maschinen?dti=0&lc=de-WW 
   // 
   // **PLC Data types**  
   //  LSicar_typeEeMenPiCalc 
   //  LSicar_typeEeMenPiEstate 
   //  LSicar_typeEeMenPiLimit 
   //  typeEnMeterOutputData 
   //  typeMeasDataProfileE3 
   //  
   // **WinCC Faceplates**  
   // 
   // ![Image](EemEnPiCalc/en/image3.PNG)
   // 
   // **WinCC Screen**  
   //  
   // ![Image](EemEnPiCalc/en/image4.PNG)
   //  
   // # Devices & networks 
   // 
   // An additional AI Energy Meter has been added and configured in the SICAR project. The user data has been  
   // configured as module version “EE@Industry measured data profile e3”.  
   // 
   // Select the module version according to your requirements. The data assignment in the FC blocks has to be adjusted according to the selected module version. 
   // 
   // ![Image](EemEnPiCalc/en/image5.PNG)
   //  
   //  
   // 
   // #### PLC Programm blocks 
   // 
   // ##### CallEnSeem  
   // The block is called in OB “CYCLIC_INTERRUPT_100MS_OB” (100ms cycle). The block contains the following instructions which can be found in “Instructions > Optional packages > Energy Suite extensions”.
   // 
   // **EnS_EEm_Calc:**  
   // The instruction calculates operating state-related energy data of machines and plants for uniform efficiency evaluation, in accordance with the VDMA 34179 measuring directive. 
   // 
   // ---
   // Note
   // :     The instruction calculates the energy efficiency value of the respective state for up to 8 operating states, and the global energy efficiency value. 
   // :     The maximum number of configurable measuring points is 10. Refer to the documentation of the entry ID. 
   // 
   // ---
   // 
   // **EnS_EEm_Report:**  
   // The instruction writes the data for the efficiency report to the data log on the SIMATIC memory card, in accordance with the VDMA 34179 measuring directive. The data log is a CSV file. 
   // 
   // #### CallEnEffMonitor
   // ---
   // Note
   // :     The assignment of the readings as well as the formation of additional signals can be represented only exemplarily here. It has to be adapted to the actual plant conditions! 
   // 
   // ---
   // 
   // * Networks 1 & 2: The readings of the two AI-Energy-Meters are entered in the DB “EeMonitor”, in an array [0..9] in accordance with the measurement data profile “typeMeasDataProfileE3”. 
   // * Network 3: According to the selection of a measuring point on the HMI, data of the respective measuring point is routed to the HMI data area. The selection is done with a Pull-Down menu and a symbolic I/O field. 
   // * Network 4: Several tags in the EnS…data types are not marked as accessible / visible. In order to display these tags on the HMI all the same, they are routed to DB “EeMonitor” in structure “typeEnMeterWorkHmi”. There the tags are marked as accessible / visible.  
   // * Network 5: A collective signal is generated, according to the exemplary calls for OP area 1. This is only an example! The collective signal shows that the plant is producing parts, by a disjunction (OR) of all outputs. If an output is controlled, the plant is moving and producing parts. This collective signal is used later on to generate the energetic states “eState”. A delay of 3 seconds has been configured so that a short break in controlling the outputs will not change the energetic state. *
   // * Network 6: The signals for the energetic states are generated here. 
   // * Network 7: Simulation On/Off: A part counter is simulated here. Note: the simulation can be switched on and off with a button in the screen. 
   // * Network 8: Simulation On/Off. Energy counters for both AI-Energy-Meters are simulated here. Note: the simulation can be switched on and off with a button in the screen. 
   // * Network 9: Call of blocks “EemDemoSimulation” and “EemDemoResetValEMeter”. 
   // * Network 10: Call of block “EemEnPiCalc” and data routing according to the selection of a measuring point on the HMI. 
   // * Network 11: Error evaluation of block “EemEnPiCalc” to generate ProDiag messages. 
   // * Network 12: Error evaluation of block “EnS_EEm_Report” to generate ProDiag messages.  
   // 
   // #### EemDemoResetValEMeter  
   // 
   // The block resets certain measurement values by controlling the respective outputs in the I/O area of the AI-Energy-Meter. 
   // 
   // #### EemDemoSimulation  
   // 
   // This block simulates higher or lower energy values, according to the energetic states “eState”. 
   // 
   // #### EemEnPiCalc
   // This block calculates the ENPI (Energy value Pro Item). It substitutes the script “EEm_EnPI_Efficiency” of the entry ID. 
   // 
   // ---
   // Note
   // :     All block parameters are provided with “pre-defined actual parameters”.
   // 
   // ---
   // 
   // **Operation mode Automatic / Manual**  
   // 
   // The blocks are independent of operation modes. Therefor they are not assigned to any operation mode area. 
   // 
   // **PLC Alarm text list**  
   // 
   // The following PLC alarm text lists have been created: 
   // 
   // * **EEMonitor_Calc_Warn_PD** ProDiag alarm text list for alarms by instruction “EnS_EEm_Calc”.   
   // * **EEMonitor_Report_Warn_PD** ProDiag alarm text list for alarms by instruction “EnS_EEm_Report”.   
   // Both PLC alarm text lists have been entered in the PLC alarm text list “GLOBAL_GENERAL_AlarmTextList”. 
   // 
   // ---
   // Note
   // :     The alarm texts are provided in two languages (German, English). Please consider the multilingual nature of the entries. 
   // 
   // ---
   // 
   // #### PLC Data types 
   // 
   // PLC data types used for PLC program block or HMI faceplate:  
   // ![Image](_Icon/reference.PNG)  See ..\Library Types\LSicar_typeEeMenPiCalc.pdf  
   // 
   // #### WinCC Objects 
   // 
   // **WinCC HMI-tags**  
   // 
   // The HMI tags are stored in the tag table “AI_EnergyMeter_EEM” in the SICAR project.  
   // 
   // **WinCC Text and graphics lists**  
   // 
   // The text list “EE-MONITOR_MEASUREPOINT” contains the texts necessary for the pull-down menu / symbolic I/O field in the screen. Please take into account the multilingual nature of the entries.  
   // 
   // **WinCC Faceplates**  
   // 
   // The faceplates are stored in the project library, in folder “types”. They have been created using several WinCC objects; they are animated depending on the state. 
   // 
   // * EEM_EnPI_EnergyPerItem:	display of ENPI (ENergy Per Item) 
   // * EEM_ViewBar_Diff-AVG-REF:	bar display to compare reference value and average value 
   // * EEM_ViewBar_EState-Total:	bar display of energy status (not used at this time) 
   // * EEM_ViewBarCurve_EState:	Total: bar display and curve display of the energy values  
   // 
   // **WinCC-screen** 
   // 
   // 1. HMI Screens:	EE-MONITOR_ENERGY: display of the energy values 
   // 2. HMI Popup-screens 
   // 	* EEM_LEGEND_Popup: 		Legend 
   // 	* EEM_INFO-MACHINE_Popup: 	Machine information 
   // 	* EEM_STARTMEASURE_Popup: 	Popup to start the normal measurement or the reference measurement  
   // 	* EEM_UIPE_Popup: 		display of voltage, current, power, and energy 
   // 	* MORE_EEM_Popup: 		Popup with additional buttons 
   // 	* MORE_AddOn_Popup: 		supplemented  with button “EE-Monitor” 
   // 
   //  
   // 
   // {.pageWidth}
   // ![Image](EemEnPiCalc/en/image6.PNG)
   //  
   //  
   // 
   // #### Additional information
   // 
   // #### Update info
   // 
   // #### Further documentations
END_REGION

REGION Network 3: EE-Monitor: "Recalc"
   // Toggeln für autom. Aktualisierung der Werte im Bild jeden zweiten Zyklus (alle 200ms) / Toggle for autom. updating the values in the screen every 2nd cycle (every 200ms)
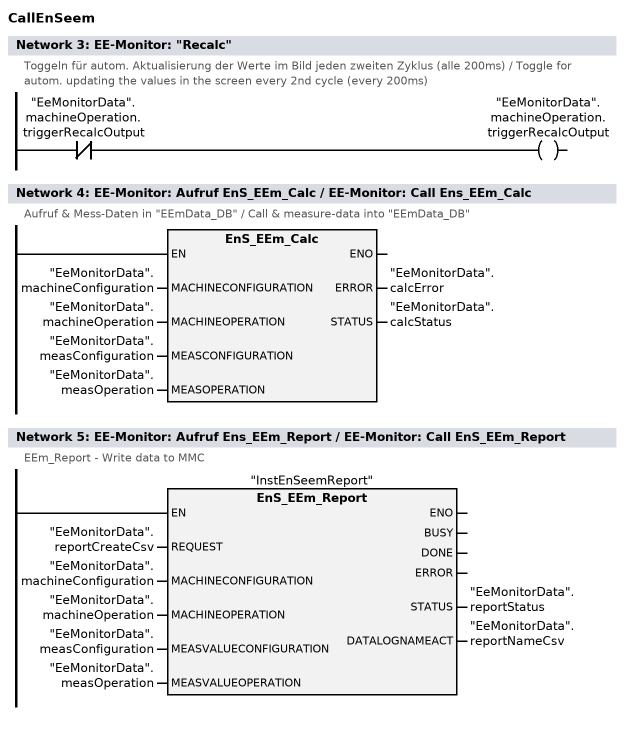
   RUNG wire#powerrail
      I_Contact( "EeMonitorData".machineOperation.triggerRecalcOutput )
      Coil( "EeMonitorData".machineOperation.triggerRecalcOutput )
   END_RUNG
   // the same network as SCL:
   "EeMonitorData".machineOperation.triggerRecalcOutput := NOT "EeMonitorData".machineOperation.triggerRecalcOutput;
END_REGION

REGION Network 4: EE-Monitor: Aufruf EnS_EEm_Calc / EE-Monitor: Call Ens_EEm_Calc
   // Aufruf & Mess-Daten in "EEmData_DB" / Call & measure-data into "EEmData_DB"
   RUNG wire#powerrail
      EnS_EEm_Calc(machineConfiguration := "EeMonitorData".machineConfiguration, machineOperation := "EeMonitorData".machineOperation, measConfiguration := "EeMonitorData".measConfiguration, measOperation := "EeMonitorData".measOperation, error => "EeMonitorData".calcError, status => "EeMonitorData".calcStatus)
   END_RUNG
   // the same network as SCL:
   EnS_EEm_Calc(machineConfiguration := "EeMonitorData".machineConfiguration,
                machineOperation := "EeMonitorData".machineOperation,
                measConfiguration := "EeMonitorData".measConfiguration,
                measOperation := "EeMonitorData".measOperation,
                error => "EeMonitorData".calcError,
                status => "EeMonitorData".calcStatus);
END_REGION

REGION Network 5: EE-Monitor: Aufruf Ens_EEm_Report / EE-Monitor: Call EnS_EEm_Report
   // EEm_Report - Write data to MMC
   RUNG wire#powerrail
      "InstEnSeemReport".EnS_EEm_Report(request := "EeMonitorData".reportCreateCsv, machineConfiguration := "EeMonitorData".machineConfiguration, machineOperation := "EeMonitorData".machineOperation, measValueConfiguration := "EeMonitorData".measConfiguration, measValueOperation := "EeMonitorData".measOperation, busy =>, done =>, error =>, status => "EeMonitorData".reportStatus, dataLogNameAct => "EeMonitorData".reportNameCsv)
   END_RUNG
   // the same network as SCL:
   "InstEnSeemReport"(request := "EeMonitorData".reportCreateCsv,   // EnS_EEm_Report
                      machineConfiguration := "EeMonitorData".machineConfiguration,
                      machineOperation := "EeMonitorData".machineOperation,
                      measValueConfiguration := "EeMonitorData".measConfiguration,
                      measValueOperation := "EeMonitorData".measOperation,
                      status => "EeMonitorData".reportStatus,
                      dataLogNameAct => "EeMonitorData".reportNameCsv);
END_REGION
END_FUNCTION

ORGANIZATION_BLOCK "ProgrammingError"   // OB121, LAD, ProgrammingError
// stored: SetENOAutomatically false
   VAR_INPUT
      BlockNr : UInt;   // Number of causing block
      Reaction : USInt;   // 0:ignore, 1:substitute, 2:skip
      Fault_ID : Byte;   // Fault identifier
      BlockType : USInt;   // 16#01:OB, 16#02:FC, 16#03:FB, 16#04:SFC, 16#05:SFB, 16#06:DB: Type of block causing the error
      Area : USInt;   // Area where the error occured
      DBNr : DB_ANY;   // DB number if Area = DB or DI
      Csg_OBNr : OB_ANY;   // Number of OB causing the error
      Csg_Prio : USInt;   // Priority of OB causing the error
      Width : USInt;   // 0:bit, 1:byte, 2:word, 3:dword, 4:lword
   END_VAR
BEGIN
END_ORGANIZATION_BLOCK

ORGANIZATION_BLOCK "Startup"   // OB100, LAD, Startup
TITLE = "Complete Restart"
// stored: AutoNumber false, IsIECCheckEnabled true, SetENOAutomatically true
   VAR_INPUT
      LostRetentive : Bool;   // True if retentive data are lost
      LostRTC : Bool;   // True if date and time are lost
   END_VAR
   VAR_TEMP
      tempError : Bool;
      tempStatus : Word;
      tempDiagnostics : "LAF_typeDiagnosticsSimple";
   END_VAR
BEGIN

REGION Network 1: Erster Zyklus bit setzen / Set first cycle bit
   // Setze das "erster Zyklus" Signal und die Signale immer EIN sowie immer AUS / Set the first cycle signal
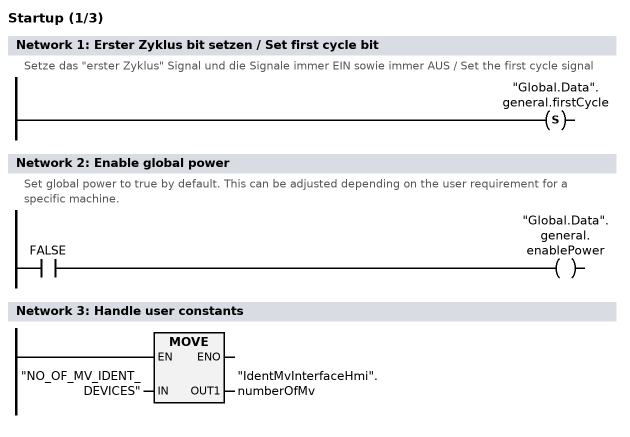
   RUNG wire#powerrail
      S_Coil( "Global.Data".general.firstCycle )
   END_RUNG
   // the same network as SCL:
   "Global.Data".general.firstCycle := TRUE;
END_REGION

REGION Network 2: Enable global power
   // Set global power to true by default. This can be adjusted depending on the user requirement for a specific machine.
   RUNG wire#powerrail
      Contact( FALSE )
      Coil( "Global.Data".general.enablePower )
   END_RUNG
   // the same network as SCL:
   "Global.Data".general.enablePower := FALSE;
END_REGION

REGION Network 3: Handle user constants
   RUNG wire#powerrail
      Move(in := "NO_OF_MV_IDENT_DEVICES", out1 => "IdentMvInterfaceHmi".numberOfMv)
   END_RUNG
   // the same network as SCL:
   "IdentMvInterfaceHmi".numberOfMv := "NO_OF_MV_IDENT_DEVICES";
END_REGION

